///Check valve position
IF iq_stValve.i_xClsLS AND  iq_stValve.i_xOpnLS THEN
    iq_stValve.eState:=INVALID;
ELSIF NOT iq_stValve.i_xClsLS AND iq_stValve.i_xOpnLS AND iq_stValve.q_xOPN_DO THEN
    iq_stValve.eState:=OPEN;
ELSIF NOT iq_stValve.i_xClsLS AND iq_stValve.i_xOpnLS AND NOT iq_stValve.q_xOPN_DO THEN
    iq_stValve.eState:=OPEN_F;
ELSIF iq_stValve.i_xClsLS AND NOT iq_stValve.i_xOpnLS AND NOT iq_stValve.q_xOPN_DO THEN
    iq_stValve.eState:=CLOSED;
ELSIF NOT iq_stValve.i_xClsLS AND NOT iq_stValve.i_xOpnLS THEN
    iq_stValve.eState:=MOVING;
ELSE
    iq_stValve.eState:=INVALID;
END_IF

// Update hysteresis
///////////////////////////////////////////////////
IF iq_stValve.rAT_VAC_SP_LAST <> iq_stValve.rAT_VAC_SP OR xFirstPass THEN
    iq_stValve.rAT_VAC_SP_LAST := iq_stValve.rAT_VAC_SP;
    iq_stValve.rAT_VAC_HYS := iq_stValve.rHYST_PERC * iq_stValve.rAT_VAC_SP;
END_IF

iq_stValve.rAT_VAC_HYS := LIMIT(0, iq_stValve.rAT_VAC_HYS, iq_stValve.rAT_VAC_SP);
IF iq_stValve.rAT_VAC_SP <> 0 THEN
    IF iq_stValve.rHYST_PERC <> (iq_stValve.rAT_VAC_HYS / iq_stValve.rAT_VAC_SP) THEN
        iq_stValve.rHYST_PERC := LIMIT(0, (iq_stValve.rAT_VAC_HYS / iq_stValve.rAT_VAC_SP) ,1);
    END_IF

END_IF
// Valve at vacuum check
///////////////////////////////////////////////////
    set := i_stUSG.rPRESS < iq_stValve.rAT_VAC_HYS AND i_stDSG.rPRESS < iq_stValve.rAT_VAC_HYS AND i_stUSG.xPRESS_OK AND i_stDSG.xPRESS_OK;
     iq_stValve.xAT_VAC S= set;
    reset := i_stUSG.rPRESS > iq_stValve.rAT_VAC_SP OR i_stDSG.rPRESS > iq_stValve.rAT_VAC_SP OR NOT i_stUSG.xPRESS_OK OR NOT i_stDSG.xPRESS_OK;
    iq_stValve.xAT_VAC R= reset;

// Differential pressure check
///////////////////////////////////////////////////
    (* Calc the differential pressure across the valve *)
    rDiffPress := ABS(i_stUSG.rPRESS - i_stDSG.rPRESS);

    (* As long as the differential pressure is less than 30mbar, the valve is allowed to open *)
    IF rDiffPress <= rDiffPressAllowed AND i_stUSG.xPRESS_OK AND i_stDSG.xPRESS_OK THEN
        iq_stValve.xDP_OK := TRUE;
    ELSE
        iq_stValve.xDP_OK	:= FALSE;
        (* If the differential pressure is exceeded, even when the valve is open,
        the state is unexpected and triggers a fault, because it suggests that something
        is wrong with the valve, or gauges or mapping or there is a major leak on one side.*)
        iq_stValve.eVGC_State := ERR_DiffPress;
    END_IF

// Valve state
///////////////////////////////////////////////////
CASE iq_stValve.eVGC_State OF
    Vented: (* The Vented state is used during pump down *)
        //Log new state
        IF ePrevState <> iq_stValve.eVGC_State THEN
            fbLogger(sMsg:='Vented', eSevr:=TcEventSeverity.Info);
            ePrevState := iq_stValve.eVGC_State;
        END_IF

        (* Assuming the pump down went well, we are now at vacuum on both sides,
        so we move to the vacuum state, otherwise remain in the vented state *)
        IF iq_stValve.xAT_VAC AND (NOT (iq_stValve.xERR_DifPres)) AND  (NOT (iq_stValve.xERR_SP)) and  (NOT (iq_stValve.xERR_ExtFault))THEN
            iq_stValve.eVGC_State := AtVacuum;
        ELSE
            iq_stValve.eVGC_State := Vented;
        END_IF

    AtVacuum:
        //Log new state
        IF ePrevState <> iq_stValve.eVGC_State THEN
            fbLogger(sMsg:='Vacuum setpoint satisfied', eSevr:=TcEventSeverity.Info);
            ePrevState := iq_stValve.eVGC_State;
        END_IF

        IF iq_stValve.xAT_VAC THEN
        (* If both pressure setpoints are made,
        then enable the differential pressure interlock, regardless of the valve state
        assuming we're using some kind of ion gauge where a pressure setpoint cannot be higher than 1E-4 T *)
        iq_stValve.eVGC_State := AtVacuum;

        ELSE

            (* If the valve is open (or in an unknown state) and either gauge is not at it's vacuum setpoint,
            we have a loss of vacuum error *)
            IF (iq_stValve.i_xOpnLS OR (NOT iq_stValve.i_xOpnLS AND NOT iq_stValve.i_xClsLS)) THEN
                iq_stValve.eVGC_State := ERR_LostVac;
                iq_stValve.xERR_SP := TRUE; //TAW changed this to the ERR_SP bool because I think that's what it was intended to be?

            (* Alternatively, if the valve is already closed and we lose pressure on one side,
            it was probably intentional venting, so we calmly move back to venting mode, and
            disable the differential pressure interlock *) //??
            ELSIF iq_stValve.i_xClsLS THEN
                iq_stValve.eVGC_State := Vented;
            END_IF

        END_IF
    ERR_DiffPress:
        //Log new state
        IF ePrevState <> iq_stValve.eVGC_State THEN
            fbLogger(sMsg:='Potential accidental vent.', eSevr:=TcEventSeverity.Critical);
            ePrevState := iq_stValve.eVGC_State;
        END_IF

        IF NOT (iq_stValve.xERR_DifPres) THEN
            iq_stValve.eVGC_State := Vented;
        END_IF


    ERR_LostVac:
        //Log new state
        IF ePrevState <> iq_stValve.eVGC_State THEN
            fbLogger(sMsg:='Unexpected loss of vacuum while valve was open.', eSevr:=TcEventSeverity.Critical);
            ePrevState := iq_stValve.eVGC_State;
        END_IF
        IF NOT (iq_stValve.xERR_SP) THEN
            iq_stValve.eVGC_State := Vented;
        END_IF

    ERR_ExtFault:
        //Log new state
        IF ePrevState <> iq_stValve.eVGC_State THEN
            fbLogger(sMsg:='Lost external interlock while valve was open.', eSevr:=TcEventSeverity.Critical);
            ePrevState := iq_stValve.eVGC_State;
        END_IF
        IF NOT (iq_stValve.xERR_ExtFault) AND (NOT i_xExt_OK) THEN
            iq_stValve.eVGC_State := Vented;
        END_IF
    END_CASE



IF (NOT i_xExt_OK) THEN
    iq_stValve.eVGC_State := ERR_ExtFault;
    iq_stValve.xERR_ExtFault := TRUE;
END_IF

// Interlock evaluation - with bypass for DP ILK bypass
///////////////////////////////////////////////
IF i_xDis_DPIlk THEN
    iq_stValve.xOPN_OK := iq_stValve.xEXT_OK; // AND iq_stValve.xDP_OK ;
ELSE
    iq_stValve.xOPN_OK := iq_stValve.xEXT_OK AND iq_stValve.xAT_VAC;
END_IF


(* Valve operation *)

(* Override logic *)
(* Goal: give ability to override, but do so in a way that people won't forget it.
Solution: Override only after ten seconds of override, protect against blips,
when the valve permission goes true for more than ten seconds consistently, remove override
*)

tonDelOK(IN:=iq_stValve.xOPN_OK, PT:=tDelOK);
rtOK(CLK:=tonDelOK.Q);
IF rtOK.Q AND iq_stValve.pv_xOvrdOpn THEN
    iq_stValve.pv_xOvrdOpn :=FALSE;
    if (iq_stValve.eState = OPEN) AND (i_xOverrideMode) THEN iq_stValve.pv_xOPN_SW := TRUE; END_IF  //for seamless transition
    //Log
    fbLogger(sMsg:='Override expired', eSevr:=TcEventSeverity.Warning);

END_IF

//Override timer
tonOvrd(IN:=iq_stValve.pv_xOvrdOpn, PT:=tOvrd);

(* If Epics Command to close the Valve, check if PMPS and EPS are ok, otherwise Keep command set to open valve *)
IF NOT(iq_stValve.pv_xOPN_SW) AND ((NOT i_xPMPS_OK) OR (NOT i_xEPS_OK)) THEN
    //iq_stValve.pv_xOPN_SW := TRUE; // plc to only reset never to set this signal
END_IF
(* Reset the EPICS command to open the valve if the interlock is lost *)
(* based on EPS ok state, EPS overrides OPN_OK*)
IF NOT iq_stValve.xOPN_OK THEN
    IF i_xEPS_OK THEN iq_stValve.pv_xOPN_SW := FALSE; iq_stValve.sErrorMessage := 'ILK Active';
    ELSE //iq_stValve.pv_xOPN_SW := TRUE;		// plc to only reset never to set this signal
    END_IF
END_IF

(* Here's where the valve opens *)
iq_stValve.q_xOPN_DO := (iq_stValve.pv_xOPN_SW AND iq_stValve.xOPN_OK) OR (tonOvrd.Q AND i_xOverrideMode);

(* When the valve  is open MPS is OK*)
xMPS_OK := i_xOpnLS XOR i_xClsLS;

///Check valve moving postion timout
IF NOT iq_stValve.i_xClsLS AND tCLStimeout.Q THEN
    iq_stValve.bErrorPresent := TRUE;
    iq_stValve.sErrorMessage := 'Close Timeout';
ELSIF NOT iq_stValve.i_xOpnLS AND tOPNtimeout.Q THEN
    iq_stValve.bErrorPresent := TRUE;
    iq_stValve.sErrorMessage := 'Open Timeout';
END_IF
IF (iq_stValve.eState=INVALID) THEN
    iq_stValve.bErrorPresent := TRUE;
    iq_stValve.sErrorMessage := CONCAT(sPath,'Invalid Valve Position');
END_IF
(*Timers*)
tOPNtimeout(IN:= iq_stValve.q_xOPN_DO, PT := tTimeOutDuration );
tCLStimeout(IN:= NOT iq_stValve.q_xOPN_DO, PT := tTimeOutDuration);


// Log valve timeouts
tErrorPresent(CLK:=iq_stValve.bErrorPresent);
IF tErrorPresent.Q THEN fbLogger(sMsg:=iq_stValve.sErrorMessage, eSevr:=TcEventSeverity.Warning); END_IF

// Log valve open
tAction(CLK:= iq_stValve.q_xOPN_DO);
IF tAction.Q THEN fbLogger(sMsg:='Valve commanded open', eSevr:=TcEventSeverity.Info); END_IF

// Log override mode enabled
tOverrideActivated(CLK:= (tonOvrd.Q AND i_xOverrideMode));
IF tOverrideActivated.Q THEN fbLogger(sMsg:='Valve override mode activated', eSevr:=TcEventSeverity.Warning); END_IF


// Alarm reset
//////////////////////////////////////
ACT_ResetAlarms();

(*IO Mapping*)
ACT_IO();

(*FAST FAULT*)
fbFF(i_xOK := xMPS_OK,
    i_xReset := i_xReset,
    i_xAutoReset :=TRUE,
    io_fbFFHWO := io_fbFFHWO);

ACTION ACT_IO:
(*inputs*)
iq_stValve.i_xOpnLS := 	i_xOpnLS;
iq_stValve.i_xClsLS:=	i_xClsLS;
iq_stValve.xEXT_OK := i_xEXT_OK;
iq_stValve.xOverrideMode := i_xOverrideMode;
(*outputs*)
q_xOPN_DO:= iq_stValve.q_xOPN_DO;
END_ACTION

ACTION ACT_ResetAlarms:
iq_stValve.xERR_DifPres R= iq_stValve.pv_xAlmRst;
iq_stValve.xERR_SP R= iq_stValve.pv_xAlmRst;
iq_stValve.bErrorPresent R= iq_stValve.pv_xAlmRst;

IF ( iq_stValve.pv_xAlmRst) THEN
    iq_stValve.sErrorMessage :='';
END_IF
END_ACTION

METHOD PUBLIC M_IsClosed : BOOL
VAR_INPUT
END_VAR
M_IsClosed := (This^.iq_stValve.eState = E_ValvePositionState.CLOSED);
END_METHOD

METHOD PUBLIC M_IsOpen : BOOL
VAR_INPUT
END_VAR
M_IsOpen := (This^.iq_stValve.eState = E_ValvePositionState.OPEN);
END_METHOD

// Use this Methode to Open or close the valve by setting the OPN_SW to the input value.
METHOD PUBLIC M_Set_OPN_SW : BOOL
VAR_INPUT
        value:BOOL;
END_VAR
This^.iq_stValve.pv_xOPN_SW := value;
END_METHOD

END_FUNCTION_BLOCK

// ---- POUs/Functions/Deprecated/Valves/FB_VGC_EBD.TcPOU
(*Deprecated*)
(* This function block is similar to the FB_VGC, except it has 2 outputs to actuate the Valve*)
(* This function block implements basic functionality for Isolation Gate Valves*)
(* This function block interlock is as follows:
1. The valve can be opened when the difference between the pressures on both sides is
less than the maximum differential pressure.
2. This rule persists until the pressures on both sides are lower than the vacuum-setpoint.
3. Once at-vac, the valve will close if the pressure on either side rises above the setpoint.*)
(*This function block also implements PMPS and EPS interlocks, as well as Fast MPS trigger*)
{attribute 'no_check'}
{attribute 'obsolete' := 'FB_VGC_EBD has been deprecated and is not valid!'}
FUNCTION_BLOCK FB_VGC_EBD
VAR_IN_OUT

END_VAR
VAR_INPUT
    (*Upstream Gauge, usually ion gauge*)
    i_stUSG	:	ST_VG;
    (*Downstream Gauge, usually ion gauge*)
    i_stDSG	:	ST_VG;
    {attribute 'pytmc' := '
    pv: Dis_DPIlk
    '}
    i_xDis_DPIlk : BOOL := FALSE;  (* Set to true when calling the function to disable the differential pressure interlock *)
    {attribute 'pytmc' := '
    pv: EPS_OK
    '}
    i_xEPS_OK:	BOOL	:= TRUE; (*External EPS interlock, Set to TRUE when no EPS interlock is required, otherwise set to correct interlock signal*)
    {attribute 'pytmc' := '
    pv: MPS_OK
    '}
    i_xPMPS_OK:	BOOL	; (*External MPS interlock, Set to TRUE when no PMPS interlock is required*)
    i_xExt_OK: BOOL; (*Other External Interlock, Set to True when no external interlock is required*)
    i_xOverrideMode : BOOL; (*To be linked to global override bit. This Overrides Vacuum logic only, EPS, MPS and PMPS are still enforces*)
    // Reset fault
    {attribute 'pytmc' := '
    pv: FF_Reset
    '}
    i_xReset: BOOL;
    i_sDevName : T_MaxString :=  'VGC'; // Device name for diagnostic
END_VAR
VAR_OUTPUT
    {attribute 'pytmc' := '
    pv:
    '}
    iq_stValve : ST_VGC; (* All valve data and states will be in this struct*)

    {attribute 'pytmc' := '
    pv: MPS_FAULT_OK
    field: ZNAM MPS FAULT ;
    field: ONAM MPS OK ;
    '}
    xMPS_OK:	BOOL; (*MPS Fast OK, is set when the Valve is Open*)
END_VAR
VAR_IN_OUT
    io_fbFFHWO    :    FB_HardwareFFOutput;
END_VAR
VAR
    // PMPS
    fbFF    :    FB_FastFault :=(
        i_DevName := 'VGC',
        i_Desc := 'Fault occurs when the valve is not in open state',
        i_TypeCode := 16#1010);
    {attribute 'instance-path'}
    {attribute 'noinit'}
    sPath: STRING;

    rDiffPressAllowed	:	REAL := 22.5; // Torr, Default value comes from Vat Valve Manual
    rDiffPress : REAL;
    set : BOOL;
    reset: BOOL;

    xFirstPass	:	BOOL;
    fbFSInit		:	R_TRIG;

    tonDelOK : TON;
    rtOK	:	R_TRIG;
    tonOvrd	:	TON;

    tDelOK	:	TIME := T#60S;
    tOvrd	:	TIME := T#10s;


    (* Timeouts*)
    tTimeOutDuration: TIME:= T#30S;
    tOPNtimeout: TON;
    tCLStimeout:TON;


     // For logging
    fbLogger : FB_LogMessage := (eSubsystem:=E_SubSystem.VACUUM);
    ePrevState : E_VGC;
    tErrorPresent : R_TRIG;
    tAction : R_TRIG; // Primary action of this device (OPN_DO, PUMP_RUN, etc.)
    tOverrideActivated : R_TRIG;

    (*IO*)
    i_xOpnLS	AT%I*: BOOL;
    i_xClsLS	AT%I*: BOOL;
    q_xOPN_DO	AT%Q*: BOOL;
    q_xOPN_DO_2	AT%Q*: BOOL;

END_VAR

(* Vacuum gate valve
A. Wallace
16-10-29

A gate valve isolates vacuum volumes. Ideally it can be opened when a system is vented
to allow for faster pumping, and will close when high vacuum is lost.

The following behavior is good for valves in something like a gas attenuator.
This function block does the following:
1. The valve can be opened when the difference between the pressures on both sides is
less than the maximum differential pressure.
2. This rule persists until the pressures on both sides are lower than the vacuum-setpoint.
3. Once at-vac, the valve will close if the pressure on either side rises above the setpoint.

Alternatively, the differential pressure interlock can be disabled so the valve may only be opened
if the pressure on both sides is lower than the at-vacuum-setpoint. You want this behavior if
the valve is to be used in a UHV section.

Hysteresis is employed to ensure a smooth transition from vented/pumping down, to at-vac.

Finally, an override system is built in so you can bypass all the interlocking logic and
get back online.
*)
(* 10/1/2018 Margaret Ghaly included EPS, PMPS Checkes and MPS trigger signals*)


fbFSInit( CLK := TRUE, Q => xFirstPass);
(*IO Mapping*)
ACT_IO();

(* On first PLC pass, put valve into vented state, which implies a closed valve *)
IF xFirstPass THEN
    iq_stValve.eVGC_State := Vented;
    iq_stValve.pv_xOPN_SW := FALSE;
    fbFF.i_DevName := i_sDevName;
END_IF


///Check valve postion
IF iq_stValve.i_xClsLS AND  iq_stValve.i_xOpnLS THEN
    iq_stValve.eState:=INVALID;
ELSIF NOT iq_stValve.i_xClsLS AND iq_stValve.i_xOpnLS AND iq_stValve.q_xOPN_DO THEN
    iq_stValve.eState:=OPEN;
ELSIF iq_stValve.i_xClsLS AND NOT iq_stValve.i_xOpnLS AND NOT iq_stValve.q_xOPN_DO THEN
    iq_stValve.eState:=CLOSED;
ELSIF NOT iq_stValve.i_xClsLS AND NOT iq_stValve.i_xOpnLS THEN
    iq_stValve.eState:=MOVING;
ELSE
    iq_stValve.eState:=INVALID;
END_IF

// Update hysteresis
///////////////////////////////////////////////////
IF iq_stValve.rAT_VAC_SP_LAST <> iq_stValve.rAT_VAC_SP OR xFirstPass THEN
    iq_stValve.rAT_VAC_SP_LAST := iq_stValve.rAT_VAC_SP;
    iq_stValve.rAT_VAC_HYS := iq_stValve.rHYST_PERC * iq_stValve.rAT_VAC_SP;
END_IF

iq_stValve.rAT_VAC_HYS := LIMIT(0, iq_stValve.rAT_VAC_HYS, iq_stValve.rAT_VAC_SP);
IF iq_stValve.rAT_VAC_SP <> 0 THEN
    IF iq_stValve.rHYST_PERC <> (iq_stValve.rAT_VAC_HYS / iq_stValve.rAT_VAC_SP) THEN
        iq_stValve.rHYST_PERC := LIMIT(0, (iq_stValve.rAT_VAC_HYS / iq_stValve.rAT_VAC_SP) ,1);
    END_IF

END_IF
// Valve at vacuum check
///////////////////////////////////////////////////
    set := i_stUSG.rPRESS < iq_stValve.rAT_VAC_HYS AND i_stDSG.rPRESS < iq_stValve.rAT_VAC_HYS AND i_stUSG.xPRESS_OK AND i_stDSG.xPRESS_OK;
     iq_stValve.xAT_VAC S= set;
    reset := i_stUSG.rPRESS > iq_stValve.rAT_VAC_SP OR i_stDSG.rPRESS > iq_stValve.rAT_VAC_SP OR NOT i_stUSG.xPRESS_OK OR NOT i_stDSG.xPRESS_OK;
    iq_stValve.xAT_VAC R= reset;

// Differential pressure check
///////////////////////////////////////////////////
    (* Calc the differential pressure across the valve *)
    rDiffPress := ABS(i_stUSG.rPRESS - i_stDSG.rPRESS);

    (* As long as the differential pressure is less than 30mbar, the valve is allowed to open *)
    IF rDiffPress <= rDiffPressAllowed AND i_stUSG.xPRESS_OK AND i_stDSG.xPRESS_OK THEN
        iq_stValve.xDP_OK := TRUE;
    ELSE
        iq_stValve.xDP_OK	:= FALSE;
        (* If the differential pressure is exceeded, even when the valve is open,
        the state is unexpected and triggers a fault, because it suggests that something
        is wrong with the valve, or gauges or mapping or there is a major leak on one side.*)
        iq_stValve.eVGC_State := ERR_DiffPress;
        iq_stValve.xERR_DifPres := TRUE;
    END_IF

// Valve state
///////////////////////////////////////////////////
CASE iq_stValve.eVGC_State OF
    Vented: (* The Vented state is used during pump down *)
        //Log new state
        IF ePrevState <> iq_stValve.eVGC_State THEN
            fbLogger(sMsg:='Vented', eSevr:=TcEventSeverity.Info);
            ePrevState := iq_stValve.eVGC_State;
        END_IF

        (* Assuming the pump down went well, we are now at vacuum on both sides,
        so we move to the vacuum state, otherwise remain in the vented state *)
        IF iq_stValve.xAT_VAC AND (NOT (iq_stValve.xERR_DifPres)) AND  (NOT (iq_stValve.xERR_SP)) and  (NOT (iq_stValve.xERR_ExtFault))THEN
            iq_stValve.eVGC_State := AtVacuum;
        ELSE
            iq_stValve.eVGC_State := Vented;
        END_IF

    AtVacuum:
        //Log new state
        IF ePrevState <> iq_stValve.eVGC_State THEN
            fbLogger(sMsg:='Vacuum setpoint satisfied', eSevr:=TcEventSeverity.Info);
            ePrevState := iq_stValve.eVGC_State;
        END_IF

        IF iq_stValve.xAT_VAC THEN
        (* If both pressure setpoints are made,
        then enable the differential pressure interlock, regardless of the valve state
        assuming we're using some kind of ion gauge where a pressure setpoint cannot be higher than 1E-4 T *)
        iq_stValve.eVGC_State := AtVacuum;

        ELSE

            (* If the valve is open (or in an unknown state) and either gauge is not at it's vacuum setpoint,
            we have a loss of vacuum error *)
            IF (iq_stValve.i_xOpnLS OR (NOT iq_stValve.i_xOpnLS AND NOT iq_stValve.i_xClsLS)) THEN
                iq_stValve.eVGC_State := ERR_LostVac;
                iq_stValve.xERR_SP := TRUE; //TAW changed this to the ERR_SP bool because I think that's what it was intended to be?

            (* Alternatively, if the valve is already closed and we lose pressure on one side,
            it was probably intentional venting, so we calmly move back to venting mode, and
            disable the differential pressure interlock *) //??
            ELSIF iq_stValve.i_xClsLS THEN
                iq_stValve.eVGC_State := Vented;
            END_IF

        END_IF

    ERR_DiffPress:
        //Log new state
        IF ePrevState <> iq_stValve.eVGC_State THEN
            fbLogger(sMsg:='Potential accidental vent.', eSevr:=TcEventSeverity.Critical);
            ePrevState := iq_stValve.eVGC_State;
        END_IF

        IF NOT (iq_stValve.xERR_DifPres) THEN
            iq_stValve.eVGC_State := Vented;
        END_IF


    ERR_LostVac:
        //Log new state
        IF ePrevState <> iq_stValve.eVGC_State THEN
            fbLogger(sMsg:='Unexpected loss of vacuum while valve was open.', eSevr:=TcEventSeverity.Critical);
            ePrevState := iq_stValve.eVGC_State;
        END_IF
        IF NOT (iq_stValve.xERR_SP) THEN
            iq_stValve.eVGC_State := Vented;
        END_IF

    ERR_ExtFault:
        //Log new state
        IF ePrevState <> iq_stValve.eVGC_State THEN
            fbLogger(sMsg:='Lost external interlock while valve was open.', eSevr:=TcEventSeverity.Critical);
            ePrevState := iq_stValve.eVGC_State;
        END_IF
        IF NOT (iq_stValve.xERR_ExtFault) AND (NOT i_xExt_OK) THEN
            iq_stValve.eVGC_State := Vented;
        END_IF
END_CASE

IF (NOT i_xExt_OK) THEN
    iq_stValve.eVGC_State := ERR_ExtFault;
    iq_stValve.xERR_ExtFault := TRUE;
END_IF

// Interlock evaluation - with bypass for DP ILK bypass
///////////////////////////////////////////////
IF i_xDis_DPIlk THEN
    iq_stValve.xOPN_OK := iq_stValve.xEXT_OK; // AND iq_stValve.xDP_OK ;
ELSE
    iq_stValve.xOPN_OK := iq_stValve.xEXT_OK AND iq_stValve.xAT_VAC;
END_IF


(* Valve operation *)

(* Override logic *)
(* Goal: give ability to override, but do so in a way that people won't forget it.
Solution: Override only after ten seconds of override, protect against blips,
when the valve permission goes true for more than ten seconds consistently, remove override
*)

tonDelOK(IN:=iq_stValve.xOPN_OK, PT:=tDelOK);
rtOK(CLK:=tonDelOK.Q);
IF rtOK.Q AND iq_stValve.pv_xOvrdOpn THEN
    iq_stValve.pv_xOvrdOpn :=FALSE;
    if (iq_stValve.eState = OPEN) AND (i_xOverrideMode) THEN iq_stValve.pv_xOPN_SW := TRUE; END_IF //for seamless transition
    //Log
    fbLogger(sMsg:='Override expired', eSevr:=TcEventSeverity.Warning);

END_IF

//Override timer
tonOvrd(IN:=iq_stValve.pv_xOvrdOpn, PT:=tOvrd);

(* If Epics Command to close the Valve, check if PMPS and EPS are ok, otherwise Keep command set to open valve *)
IF NOT(iq_stValve.pv_xOPN_SW) AND ((NOT i_xPMPS_OK) OR (NOT i_xEPS_OK)) THEN
    //iq_stValve.pv_xOPN_SW := TRUE; // plc to only reset never to set this signal
END_IF
(* Reset the EPICS command to open the valve if the interlock is lost *)
(* based on EPS ok state, EPS overrides OPN_OK*)
IF NOT iq_stValve.xOPN_OK THEN
    IF i_xEPS_OK THEN iq_stValve.pv_xOPN_SW := FALSE; iq_stValve.sErrorMessage := 'ILK Active';
    ELSE //iq_stValve.pv_xOPN_SW := TRUE;		// plc to only reset never to set this signal
    END_IF
END_IF

(* Here's where the valve opens *)
iq_stValve.q_xOPN_DO := (iq_stValve.pv_xOPN_SW AND iq_stValve.xOPN_OK) OR (tonOvrd.Q AND i_xOverrideMode);

(* When the valve  is open MPS is OK*)
xMPS_OK := (iq_stValve.eState=OPEN) OR (iq_stValve.eState=OPEN_F);//iq_stValve.i_xOpnLS;

///Check valve moving postion timout
IF NOT iq_stValve.i_xClsLS AND tCLStimeout.Q THEN
    iq_stValve.bErrorPresent := TRUE;
    iq_stValve.sErrorMessage := ' Close Timeout';
ELSIF NOT iq_stValve.i_xOpnLS AND tOPNtimeout.Q THEN
    iq_stValve.bErrorPresent := TRUE;
    iq_stValve.sErrorMessage := ' Open Timeout';
END_IF
IF (iq_stValve.eState=INVALID) THEN
    iq_stValve.bErrorPresent := TRUE;
    iq_stValve.sErrorMessage := CONCAT(sPath,' Invalid Valve Position');
END_IF


(*Timers*)
tOPNtimeout(IN:= iq_stValve.q_xOPN_DO, PT := tTimeOutDuration );
tCLStimeout(IN:= NOT iq_stValve.q_xOPN_DO, PT := tTimeOutDuration);

// Log valve timeouts
tErrorPresent(CLK:=iq_stValve.bErrorPresent);
IF tErrorPresent.Q THEN fbLogger(sMsg:=iq_stValve.sErrorMessage, eSevr:=TcEventSeverity.Warning); END_IF

// Log valve open
tAction(CLK:= iq_stValve.q_xOPN_DO);
IF tAction.Q THEN fbLogger(sMsg:='Valve commanded open', eSevr:=TcEventSeverity.Info); END_IF

// Log override mode enabled
tOverrideActivated(CLK:= (tonOvrd.Q AND i_xOverrideMode));
IF tOverrideActivated.Q THEN fbLogger(sMsg:='Valve override mode activated', eSevr:=TcEventSeverity.Warning); END_IF

// Alarm reset
//////////////////////////////////////
ACT_ResetAlarms();

(*IO Mapping*)
ACT_IO();

(*FAST FAULT*)
fbFF(i_xOK := xMPS_OK,
    i_xReset := i_xReset,
    i_xAutoReset :=TRUE,
    io_fbFFHWO := io_fbFFHWO);

ACTION ACT_IO:
(*inputs*)
iq_stValve.i_xOpnLS := 	i_xOpnLS;
iq_stValve.i_xClsLS:=	i_xClsLS;
iq_stValve.xEXT_OK := i_xEXT_OK;
iq_stValve.xOverrideMode := i_xOverrideMode;
(*outputs*)
q_xOPN_DO:= iq_stValve.q_xOPN_DO;
q_xOPN_DO_2:= iq_stValve.q_xOPN_DO;


(*ILK Devices*)
iq_stValve.sIlkUSDeviceName := This^.i_stUSG.sPath;
iq_stValve.sIlkDSDeviceName := This^.i_stDSG.sPath;
END_ACTION

ACTION ACT_ResetAlarms:
iq_stValve.xERR_DifPres R= iq_stValve.pv_xAlmRst;
iq_stValve.xERR_SP R= iq_stValve.pv_xAlmRst;
iq_stValve.bErrorPresent R= iq_stValve.pv_xAlmRst;

IF ( iq_stValve.pv_xAlmRst) THEN
    iq_stValve.sErrorMessage :='';
END_IF
END_ACTION

METHOD PUBLIC M_IsClosed : BOOL
VAR_INPUT
END_VAR
M_IsClosed := (This^.iq_stValve.eState = E_ValvePositionState.CLOSED);
END_METHOD

METHOD PUBLIC M_IsOpen : BOOL
VAR_INPUT
END_VAR
M_IsOpen := (This^.iq_stValve.eState = E_ValvePositionState.OPEN);
END_METHOD

// Use this Methode to Open or close the valve by setting the OPN_SW to the input value.
METHOD PUBLIC M_Set_OPN_SW : BOOL
VAR_INPUT
        value:BOOL;
END_VAR
This^.iq_stValve.pv_xOPN_SW := value;
END_METHOD

END_FUNCTION_BLOCK

// ---- POUs/Functions/Gauges/FB_901_ECAT.TcPOU
(* works for 901 with Ethercat interface*)
{attribute 'no_check'}
FUNCTION_BLOCK FB_901_ECAT  EXTENDS FB_GaugeBase
VAR_INPUT
END_VAR
VAR_OUTPUT
    {attribute 'pytmc' := '
    pv:
    '}
    PG	: ST_VG;
END_VAR
VAR_IN_OUT

END_VAR
VAR
    bInit: BOOL:= TRUE;(*IO*)
    xPress_OK AT%I* : BOOL;
    xOverrange AT%I* : BOOL;
    xUnderrange AT%I* : BOOL;
    i_iPRESS_R AT%I* : REAL; // input Pressure // Link to analog Input
    bWcstate AT%I* : BOOL; // 0: date valid, 1: date invalid

END_VAR

(* Standard MKS 9XX series conversion *)
(* works for 901 with Ethercat interface*)
// no div by zero
PG.rPRESS :=i_iPRESS_R;
PG.xPRESS_OK := xPress_OK and NOT bWcstate ;
IF xPress_OK and NOT bWcstate THEN
    PG.xPRESS_OK := TRUE;
    PG.eState := Valid; //Press OK
ELSIF xOverrange and NOT bWcstate THEN
    PG.xPRESS_OK := FALSE;
    PG.eState := OoR;
ELSIF xUnderrange and NOT bWcstate THEN
    PG.xPRESS_OK := FALSE;
    PG.eState := PressInvalid;

END_IF



(*Logger*)
ACT_Logger();
(* Soft IO Mapping*)
ACT_IO();

ACTION ACT_Init:
IF (bInit) THEN
    bInit := False;

    //set pressure units to Torr
    // value 0x00A10000 SDO index 0xf840, si 0x01 UDINT
END_IF
END_ACTION

ACTION ACT_IO:

IF PG.xPRESS_OK THEN
      PG.i_iPRESS_R := REAL_TO_INT(i_iPRESS_R);
ELSE
    PG.rPRESS := 0.0;
END_IF
PG.sPath := sPath;
END_ACTION

ACTION ACT_Logger:

//STATE Logger
IF ePrevState <> PG.eState THEN
      CASE PG.eState OF
        ValidHi:
            fbLogger(sMsg:='Gauge pressure valid high.', eSevr:=TcEventSeverity.Info);
        ValidLo:
            fbLogger(sMsg:='Gauge pressure valid low.', eSevr:=TcEventSeverity.Info);
        Valid:
            fbLogger(sMsg:='Gauge pressure valid.', eSevr:=TcEventSeverity.Info);
          GaugeDisconnected:
            fbLogger(sMsg:='Gauge Disconnected.', eSevr:=TcEventSeverity.Critical);
        PressInvalid:
            fbLogger(sMsg:='Gauge pressure invalid.', eSevr:=TcEventSeverity.Warning);
        OoR:
            fbLogger(sMsg:='Gauge pressure out of range.', eSevr:=TcEventSeverity.Warning);
        Starting:
            fbLogger(sMsg:='Gauge starting.', eSevr:=TcEventSeverity.Info);
      END_CASE
      ePrevState := PG.eState;
  END_IF
END_ACTION

END_FUNCTION_BLOCK

// ---- POUs/Functions/Gauges/FB_9XX.TcPOU
(* Standard MKS 9XX series conversion *)
(* works for 925 *)
FUNCTION_BLOCK FB_9XX EXTENDS FB_GaugeBase
VAR_INPUT
END_VAR
VAR_OUTPUT
    {attribute 'pytmc' := '
    pv:
    '}
    PG	: ST_VG;
END_VAR
VAR_IN_OUT
END_VAR
VAR
    rV : REAL;
    fbGaugeState : FB_PressureState;
    rMaxPressure	:	REAL := 760; //Torr
    rMinPressure	:	REAL := 1E-5; //Torr
    rVMin : REAL:= 0.9;

    iTermBits: UINT := 30518 ; // The terminal's maximum value in bits default el3174 as per vacuum architecture
    (*IO*)
    i_iPRESS_R AT%I* :INT; // input Pressure // Link to analog Input
END_VAR

VAR CONSTANT
    (*Default set point 50 mT*)
    rDefaultVAC_SP: REAL := 5E-2;
END_VAR

(* Standard MKS 9XX series conversion *)
(* works for 972 and 925 *)


//Default setpoint
IF PG.rVAC_SP = 0 THEN
    PG.rVAC_SP := rDefaultVAC_SP;
END_IF
// check no div by zero
If (iTermBits=0) THEN iTermBits := 30518;END_IF
rV := 10*INT_TO_REAL(PG.i_iPRESS_R)/iTermBits;

IF rV >=rVMin THEN
    IF rV >= rVMin AND rV <= 1 THEN
        PG.rPRESS := 1E-5;
    ELSE
        PG.rPRESS := LREAL_TO_REAL(EXPT(10, rV-6));
    END_IF
    PG.xPRESS_OK := TRUE;
    PG.eState := Valid;
ELSE
    PG.xPRESS_OK := FALSE;
    IF (rV = 0) THEN PG.eState := GaugeDisconnected;
        ELSE  PG.eState := PressInvalid;
    END_IF
END_IF

(* Setpoint evaluation *)
PG.xAT_VAC := PG.xPRESS_OK AND (PG.rPRESS < PG.rVAC_SP);


(*Logger*)
ACT_Logger();
(*Soft IO Mapping*)
ACT_IO();

ACTION ACT_IO:
PG.i_iPRESS_R :=i_iPRESS_R;
PG.sPath := sPath;
END_ACTION

ACTION ACT_Logger:

//STATE Logger
IF ePrevState <> PG.eState THEN
      CASE PG.eState OF
        ValidHi:
            fbLogger(sMsg:='Gauge pressure valid high.', eSevr:=TcEventSeverity.Info);
        ValidLo:
            fbLogger(sMsg:='Gauge pressure valid low.', eSevr:=TcEventSeverity.Info);
        Valid:
            fbLogger(sMsg:='Gauge pressure valid.', eSevr:=TcEventSeverity.Info);
          GaugeDisconnected:
            fbLogger(sMsg:='Gauge Disconnected.', eSevr:=TcEventSeverity.Critical);
        PressInvalid:
            fbLogger(sMsg:='Gauge pressure invalid.', eSevr:=TcEventSeverity.Warning);
        OoR:
            fbLogger(sMsg:='Gauge pressure out of range.', eSevr:=TcEventSeverity.Warning);
        Starting:
            fbLogger(sMsg:='Gauge starting.', eSevr:=TcEventSeverity.Info);
      END_CASE
      ePrevState := PG.eState;
  END_IF
END_ACTION

METHOD M_SetBits : BOOL
VAR_INPUT
    TermBits : UINT; // The terminal's maximum value in bits
END_VAR
This^.iTermBits := TermBits;
END_METHOD

END_FUNCTION_BLOCK

// ---- POUs/Functions/Gauges/FB_972.TcPOU
{attribute 'no_check'}
FUNCTION_BLOCK FB_972  EXTENDS FB_GaugeBase
VAR_INPUT
END_VAR
VAR_OUTPUT
    {attribute 'pytmc' := '
    pv:
    '}
    PG	: ST_VG;
END_VAR
VAR_IN_OUT

END_VAR
VAR
    rV : REAL;
    iTermBits: UINT := 32767 ; // The terminal's maximum value in bits
    (*IO*)
    i_iPRESS_R AT%I* :INT; // input Pressure // Link to analog Input
END_VAR

(* Standard MKS 9XX series conversion *)
(* works for 972 and 925 *)
// no div by zero
If (iTermBits=0) THEN iTermBits := 32767;END_IF
rV := 10*INT_TO_REAL(PG.i_iPRESS_R)/iTermBits;

IF (rV > 1) AND (rV <= 7) THEN
    PG.rPRESS := LREAL_TO_REAL(EXPT(10, 2*rV-11));
    PG.xPRESS_OK := TRUE;
    PG.eState := Valid; //Press OK
ELSE
    PG.xPRESS_OK := FALSE;
    IF (rV <= 1) THEN PG.eState := GaugeDisconnected;
        ELSE PG.eState := OoR;
    END_IF
END_IF

(* Setpoint evaluation *)
PG.xAT_VAC := PG.xPRESS_OK AND (PG.rPRESS < PG.rVAC_SP);

(*Logger*)
ACT_Logger();
(* Soft IO Mapping*)
ACT_IO();

ACTION ACT_IO:
PG.i_iPRESS_R :=i_iPRESS_R;
PG.sPath := sPath;
END_ACTION

ACTION ACT_Logger:

//STATE Logger
IF ePrevState <> PG.eState THEN
      CASE PG.eState OF
        ValidHi:
            fbLogger(sMsg:='Gauge pressure valid high.', eSevr:=TcEventSeverity.Info);
        ValidLo:
            fbLogger(sMsg:='Gauge pressure valid low.', eSevr:=TcEventSeverity.Info);
        Valid:
            fbLogger(sMsg:='Gauge pressure valid.', eSevr:=TcEventSeverity.Info);
          GaugeDisconnected:
            fbLogger(sMsg:='Gauge Disconnected.', eSevr:=TcEventSeverity.Critical);
        PressInvalid:
            fbLogger(sMsg:='Gauge pressure invalid.', eSevr:=TcEventSeverity.Warning);
        OoR:
            fbLogger(sMsg:='Gauge pressure out of range.', eSevr:=TcEventSeverity.Warning);
        Starting:
            fbLogger(sMsg:='Gauge starting.', eSevr:=TcEventSeverity.Info);
      END_CASE
      ePrevState := PG.eState;
  END_IF
END_ACTION

METHOD M_SetBits : BOOL
VAR_INPUT
    TermBits : UINT; // The terminal's maximum value in bits
END_VAR
This^.iTermBits := TermBits;
END_METHOD

END_FUNCTION_BLOCK

// ---- POUs/Functions/Gauges/FB_IE514.TcPOU
(*This function is for the IE514 connected to controller IM540*)
(*This function provides ILK and Set Point Protection for the IE514*)
FUNCTION_BLOCK FB_IE514 EXTENDS FB_GaugeBase
VAR_IN_OUT
END_VAR
VAR_INPUT
    PG : ST_VG;
END_VAR
VAR_OUTPUT
    {attribute 'pytmc' := '
        pv:01
    '}
    IG_CH1 : ST_VG;
    {attribute 'pytmc' := '
        pv:02
    '}
    IG_CH2 : ST_VG;
END_VAR
VAR
    rV_CH1 : REAL; //Raw value in volts for CH1 calculated from iTermBits
    rV_CH2 : REAL; //Raw value in volts for CH2 calculated from iTermBits

    tHvDis_CH1 : TON := (PT := T#20S); //HV turn on timer
    tHvDis_CH2 : TON := (PT := T#20S); //HV turn on timer

    rtHvSw_CH1 : R_TRIG;
    rtHvSw_CH2 : R_TRIG;

    tAction_CH1 : R_TRIG;
    tAction_CH2 : R_TRIG;

    ePrevStateIG_CH1 : E_PressureState;
    ePrevStateIG_CH2 : E_PressureState;

    //rDefaultVAC_SP: REAL := 9E-3; // as per manual

    iTermBits : UINT := 30518; // The terminal's maximum value in bits default el3174 as per vacuum architecture
    binit : BOOL := TRUE;  // Do something at startup

    (*IOs to be linked*)
    /// Controls and I/Os
    i_iPRESS_R_CH1 AT %I* : INT; // input raw pressure in bits CH1 (ADC) // 'TcLinkTo' (EL3174) ^Input
    i_iPRESS_R_CH2 AT %I* : INT; // input raw pressure in bits CH2 (ADC) // 'TcLinkTo' (EL3174) ^Input
    q_xHV_DIS_CH1 AT %Q* : BOOL; // Enable Gauge High Voltage on CH1 when True // 'TcLinkTo' (EL2124) ^Output
    q_xHV_DIS_CH2 AT %Q* : BOOL; // Enable Gauge High Voltage on CH2 when True // 'TcLinkTo' (EL2124) ^Output
    i_xHV_ON AT %I*	: BOOL; // True when EMI is on  // 'TcLinkTo' (EL1004 or EL1008) ^Input
    i_xERR_CH1 AT %I* : BOOL; // TRUE when NO error is present on assigned channel
    i_xERR_CH2 AT %I* : BOOL; // TRUE when NO error is present on assigned channel
    i_xCH2_SEL AT %I* : BOOL; // TRUE when CH2 selected, FALSE when CH1 selected
END_VAR
VAR CONSTANT
    cMaxPressure : REAL := 7.5E-5; //Torr
    cMinPressure : REAL := 7.5E-14; //Torr
    cGaugeMinVoltage : REAL := 1.111; //minimum voltage corresponds to 7.5E-13 (7.498E-13)Torr which should be the minimum pressure IE514 can read.
    cGaugeMaxVoltage : REAL := 10.0; //maximum voltage corresponds 7.5E-5 Torr which should be the maximum pressure IE514 can read.
    cGaugeDisconnected : REAL := 10.2; //voltage when gauge is disconnected.
    cGaugeOff : REAL := 10.2; //voltage when gauge is turned off
    cDeadband : REAL := 0.05; //deadband in voltage
END_VAR
VAR PERSISTENT
    //Persistent variables for CH1
    rVAC_SP_CH1 : REAL;
    rPRO_SP_CH1 : REAL;
    rHYS_PR_CH1 : REAL;
    //Persistent variables for CH2
    rVAC_SP_CH2 : REAL;
    rPRO_SP_CH2 : REAL;
    rHYS_PR_CH2 : REAL;
END_VAR

(* 2-6-2023, Janez Govednik *)
(* This function will read the pressure from an IE514 gauge on an IM540. *)

(*Only ONE channel can be turned ON at the same time*)
rtHvSw_CH1(CLK := IG_CH1.xHV_SW);
rtHvSw_CH2(CLK := IG_CH2.xHV_SW);
IF rtHvSw_CH1.Q THEN
    IG_CH2.xHV_SW := FALSE;
    IG_CH2.q_xHV_DIS := FALSE;
END_IF

IF rtHvSw_CH2.Q THEN
    IG_CH1.xHV_SW := FALSE;
    IG_CH1.q_xHV_DIS := FALSE;
END_IF

//Start timers when HV ON signal triggered
tHvDis_CH1(IN := IG_CH1.q_xHV_DIS, Q => IG_CH1.xTurnOnTime);
tHvDis_CH2(IN := IG_CH2.q_xHV_DIS, Q => IG_CH2.xTurnOnTime);

(*Raw voltage conversion*)
//check no div by zero
IF (iTermBits = 0) THEN iTermBits := 30518; END_IF
rV_CH1 := 10*INT_TO_REAL(i_iPRESS_R_CH1)/iTermBits;
rV_CH2 := 10*INT_TO_REAL(i_iPRESS_R_CH2)/iTermBits;

(*RAW voltage to Pressure conversion*)
IG_CH1.rPRESS := LREAL_TO_REAL(EXPT(10, rV_CH1/10*LOG(cMaxPressure/cMinPressure) + LOG(cMinPressure))); //manual page 70 IM540 (Mode Full), (Scale) = Log
IG_CH2.rPRESS := LREAL_TO_REAL(EXPT(10, rV_CH2/10*LOG(cMaxPressure/cMinPressure) + LOG(cMinPressure))); //manual page 70 IM540 (Mode Full), (Scale) = Log

(*Pressure gauge State checks*)
//CH1
IF NOT i_xCH2_SEL AND IG_CH1.xHV_SW THEN
    IF NOT i_xERR_CH1 THEN
        IG_CH1.eState := GaugeDisconnected;
        IG_CH1.rPRESS := 0;
    ELSIF rV_CH1 <= cGaugeMaxVoltage AND rV_CH1 >= cGaugeMinVoltage AND IG_CH1.i_xHV_ON THEN
        IG_CH1.eState := Valid; // NORMAL
    ELSIF rV_CH1 >= 0.0 AND rV_CH1 < cGaugeMinVoltage AND IG_CH1.i_xHV_ON THEN
        IG_CH1.eState := OoR; //Out of range according to manual
    ELSIF rV_CH1 > cGaugeMaxVoltage AND rV_CH1 < (cGaugeMaxVoltage + cDeadband) AND IG_CH1.i_xHV_ON THEN
        IG_CH1.eState := OoR; //Out of range according to manual
    ELSIF rV_CH1 > (cGaugeMaxVoltage + cDeadband) AND tHvDis_CH1.Q THEN
        IG_CH1.eState := GaugeDisconnected; //gauge disconnected
        IG_CH1.rPRESS := 0;
    ELSIF rV_CH1 > (cGaugeMaxVoltage + cDeadband) AND NOT tHvDis_CH1.Q THEN
        IG_CH1.eState := Starting; //gauge is starting
        IG_CH1.rPRESS := 0;
    ELSE
        IG_CH1.eState := PressInvalid; //other fault - could be no gauge, controller powering up etc.
        IG_CH1.rPRESS := 0;
    END_IF
ELSE
    IG_CH1.eState := Off; // Gauge turned OFF
    IG_CH1.rPRESS := 0;
END_IF

//CH2
IF i_xCH2_SEL AND IG_CH2.xHV_SW THEN
    IF NOT i_xERR_CH2 THEN
        IG_CH2.eState := GaugeDisconnected;
        IG_CH2.rPRESS := 0;
    ELSIF rV_CH2 <= cGaugeMaxVoltage AND rV_CH2 >= cGaugeMinVoltage AND IG_CH2.i_xHV_ON THEN
        IG_CH2.eState := Valid; // NORMAL
    ELSIF rV_CH2 >= 0.0 AND rV_CH2 < cGaugeMinVoltage AND IG_CH2.i_xHV_ON THEN
        IG_CH2.eState := OoR; //Out of range according to manual
    ELSIF rV_CH2 > cGaugeMaxVoltage AND rV_CH2 < (cGaugeMaxVoltage + cDeadband) AND IG_CH2.i_xHV_ON THEN
        IG_CH2.eState := OoR; //Out of range according to manual
    ELSIF rV_CH2 > (cGaugeMaxVoltage + cDeadband) AND tHvDis_CH2.Q THEN
        IG_CH2.eState := GaugeDisconnected; //gauge disconnected
        IG_CH2.rPRESS := 0;
    ELSIF rV_CH2 > (cGaugeMaxVoltage + cDeadband) AND NOT tHvDis_CH2.Q THEN
        IG_CH2.eState := Starting; //gauge is starting
        IG_CH2.rPRESS := 0;
    ELSE
        IG_CH2.eState := PressInvalid; //other fault - could be no gauge, controller powering up etc.
        IG_CH2.rPRESS := 0;
    END_IF
ELSE
    IG_CH2.eState := Off; // Gauge turned OFF
    IG_CH2.rPRESS := 0;
END_IF

(* Ion Gauge Protection Functions *)
(* If the PG pressure is greater than the VG.PRO_SP then the gauge is disabled *)
(* If the PG pressure is less than the VG.PRO_SP then the gauge is enabled *)
(* This FB also implements some hysteresis so the gauge doesn't have rapid power cycling while near the turn on boundary *)

//CH1
IF (PG.rPRESS <= IG_CH1.rPRO_SP) AND PG.xPRESS_OK THEN
    IG_CH1.q_xHV_DIS := IG_CH1.xHV_SW;
    IG_CH1.xILKOk := TRUE;
ELSIF IG_CH1.q_xHV_DIS AND tHvDis_CH1.Q THEN
    IF IG_CH1.rPRESS > (IG_CH1.rPRO_SP + IG_CH1.rHYS_PR) OR PG.rPRESS > (IG_CH1.rPRO_SP + IG_CH1.rHYS_PR) THEN
        IG_CH1.q_xHV_DIS := FALSE;
        IG_CH1.xHV_SW := FALSE;
    END_IF
    //Adding this line because in case of interlocking gauge with another GCC or GHC PG.rPRESS value become 0 when turning it off
    IF PG.rPRESS = 0 AND NOT PG.xPRESS_OK THEN
        IG_CH1.q_xHV_DIS := FALSE;
        IG_CH1.xHV_SW := FALSE;
    END_IF
ELSE
    IG_CH1.q_xHV_DIS := FALSE;
    IG_CH1.xHV_SW := FALSE;
    IG_CH1.xILKOk := FALSE;
END_IF

//CH2
IF (PG.rPRESS <= IG_CH2.rPRO_SP) AND PG.xPRESS_OK THEN
    IG_CH2.q_xHV_DIS := IG_CH2.xHV_SW;
    IG_CH2.xILKOk := TRUE;
ELSIF IG_CH2.q_xHV_DIS AND tHvDis_CH2.Q THEN
    IF IG_CH2.rPRESS > (IG_CH2.rPRO_SP + IG_CH2.rHYS_PR) OR PG.rPRESS > (IG_CH2.rPRO_SP + IG_CH2.rHYS_PR) THEN
        IG_CH2.q_xHV_DIS := FALSE;
        IG_CH2.xHV_SW := FALSE;
    END_IF
    //Adding this line because in case of interlocking gauge with another GCC or GHC PG.rPRESS value become 0 when turning it off
    IF PG.rPRESS = 0 AND NOT PG.xPRESS_OK THEN
        IG_CH2.q_xHV_DIS := FALSE;
        IG_CH2.xHV_SW := FALSE;
    END_IF
ELSE
    IG_CH2.q_xHV_DIS := FALSE;
    IG_CH2.xHV_SW := FALSE;
    IG_CH2.xILKOk := FALSE;
END_IF


(*Pressure gauge OK checks, Backwards compatibility*)
IG_CH1.xPRESS_OK := ((IG_CH1.eState = Valid) OR IG_CH1.xBAKEOUT);
IG_CH2.xPRESS_OK := ((IG_CH2.eState = Valid) OR IG_CH2.xBAKEOUT);

(*Setpoint evaluation*)
IG_CH1.xAT_VAC := IG_CH1.xPRESS_OK AND IG_CH1.rPRESS < IG_CH1.rVAC_SP;
IG_CH2.xAT_VAC := IG_CH2.xPRESS_OK AND IG_CH2.rPRESS < IG_CH2.rVAC_SP;

(*Logger*)
ACT_Logger();

(*Soft IO Linking*)
IO();

(*Load or save the persistent variables*)
ACT_Persistent();

ACTION ACT_Logger:
// ILK logger
(*CH1 of IM540 Controller*)
IF (IG_CH1.xLog) THEN
    IF NOT IG_CH1.xILKOk AND IG_CH1.q_xHV_DIS THEN
            fbLogger(sMsg:='Lost external interlock while gauge(CH1) was on.', eSevr:=TcEventSeverity.Critical);
    END_IF

    // Log Action
    tAction_CH1(CLK := IG_CH1.xHV_SW);
    IF tAction_CH1.Q THEN fbLogger(sMsg:='Ion gauge(CH1) commanded to switch on', eSevr:=TcEventSeverity.Info); END_IF

    //STATE Logger
    IF ePrevStateIG_CH1 <> IG_CH1.eState THEN
          CASE IG_CH1.eState OF
            ValidHi:
                fbLogger(sMsg:='Gauge(CH1) pressure valid high.', eSevr:=TcEventSeverity.Info);
            ValidLo:
                fbLogger(sMsg:='Gauge(CH1) pressure valid low.', eSevr:=TcEventSeverity.Info);
            Valid:
                fbLogger(sMsg:='Gauge(CH1) pressure valid.', eSevr:=TcEventSeverity.Info);
            GaugeDisconnected:
                fbLogger(sMsg:='Gauge(CH1) Disconnected.', eSevr:=TcEventSeverity.Critical);
            PressInvalid:
                fbLogger(sMsg:='Gauge(CH1) pressure invalid.', eSevr:=TcEventSeverity.Warning);
            OoR:
                fbLogger(sMsg:='Gauge(CH1) pressure out of range.', eSevr:=TcEventSeverity.Warning);
            Starting:
                fbLogger(sMsg:='Gauge(CH1) starting.', eSevr:=TcEventSeverity.Info);
          END_CASE
          ePrevStateIG_CH1 := IG_CH1.eState;
      END_IF
END_IF

(*CH2 of IM540 Controller*)
IF (IG_CH2.xLog) THEN
    IF NOT IG_CH2.xILKOk AND IG_CH2.q_xHV_DIS THEN
            fbLogger(sMsg:='Lost external interlock while gauge(CH2) was on.', eSevr:=TcEventSeverity.Critical);
    END_IF

    // Log Action
    tAction_CH2(CLK := IG_CH2.xHV_SW);
    IF tAction_CH2.Q THEN fbLogger(sMsg:='Ion gauge(CH2) commanded to switch on', eSevr:=TcEventSeverity.Info); END_IF

    //STATE Logger
    IF ePrevStateIG_CH2 <> IG_CH2.eState THEN
          CASE IG_CH2.eState OF
            ValidHi:
                fbLogger(sMsg:='Gauge(CH2) pressure valid high.', eSevr:=TcEventSeverity.Info);
            ValidLo:
                fbLogger(sMsg:='Gauge(CH2) pressure valid low.', eSevr:=TcEventSeverity.Info);
            Valid:
                fbLogger(sMsg:='Gauge(CH2) pressure valid.', eSevr:=TcEventSeverity.Info);
            GaugeDisconnected:
                fbLogger(sMsg:='Gauge(CH2) Disconnected.', eSevr:=TcEventSeverity.Critical);
            PressInvalid:
                fbLogger(sMsg:='Gauge(CH2) pressure invalid.', eSevr:=TcEventSeverity.Warning);
            OoR:
                fbLogger(sMsg:='Gauge(CH2) pressure out of range.', eSevr:=TcEventSeverity.Warning);
            Starting:
                fbLogger(sMsg:='Gauge(CH2) starting.', eSevr:=TcEventSeverity.Info);
          END_CASE
          ePrevStateIG_CH2 := IG_CH2.eState;
      END_IF
END_IF
END_ACTION

ACTION ACT_Persistent:
(*On first PLC pass, load the persistent value into the structrue variable*)
IF (SUPER^.bRestorePersistentData) THEN
    SUPER^.bRestorePersistentData := FALSE;
    //CH1
    IF (rVAC_SP_CH1 <> 0) THEN
        IG_CH1.rVAC_SP := rVAC_SP_CH1;
    END_IF;
    IF (rPRO_SP_CH1 <> 0) THEN
        IG_CH1.rPRO_SP := rPRO_SP_CH1;
    END_IF;
    IF (rHYS_PR_CH1 <> 0) THEN
        IG_CH1.rHYS_PR := rHYS_PR_CH1;
    END_IF;
    //CH2
    IF (rVAC_SP_CH2 <> 0) THEN
        IG_CH2.rVAC_SP := rVAC_SP_CH2;
    END_IF;
    IF (rPRO_SP_CH2 <> 0) THEN
        IG_CH2.rPRO_SP := rPRO_SP_CH2;
    END_IF;
    IF (rHYS_PR_CH2 <> 0) THEN
        IG_CH2.rHYS_PR := rHYS_PR_CH2;
    END_IF;
END_IF
(*Check if a new value has been written in the structure variable copy it to the persistent variable*)
//CH1
IF NOT (IG_CH1.rVAC_SP = rVAC_SP_CH1)  THEN
    rVAC_SP_CH1 := IG_CH1.rVAC_SP;
END_IF;

IF NOT (IG_CH1.rPRO_SP = rPRO_SP_CH1) THEN
    rPRO_SP_CH1 := IG_CH1.rPRO_SP;
END_IF;

IF NOT (IG_CH1.rHYS_PR = rHYS_PR_CH1) THEN
    rHYS_PR_CH1 := IG_CH1.rHYS_PR;
END_IF;

//CH2
IF NOT (IG_CH2.rVAC_SP = rVAC_SP_CH2)  THEN
    rVAC_SP_CH2 := IG_CH2.rVAC_SP;
END_IF;

IF NOT (IG_CH2.rPRO_SP = rPRO_SP_CH2) THEN
    rPRO_SP_CH2 := IG_CH2.rPRO_SP;
END_IF;

IF NOT (IG_CH2.rHYS_PR = rHYS_PR_CH2) THEN
    rHYS_PR_CH2 := IG_CH2.rHYS_PR;
END_IF;
END_ACTION

ACTION IO:
(*soft link inputs*)
IF NOT i_xCH2_SEL THEN
    IG_CH1.i_xHV_ON := i_xHV_ON;
    IG_CH2.i_xHV_ON := FALSE;
ELSE
    IG_CH1.i_xHV_ON := FALSE;
    IG_CH2.i_xHV_ON := i_xHV_ON;
END_IF

IG_CH1.i_iPRESS_R := i_iPRESS_R_CH1;
IG_CH2.i_iPRESS_R := i_iPRESS_R_CH2;

(*soft link outputs*)
q_xHV_DIS_CH1 := IG_CH1.q_xHV_DIS;
q_xHV_DIS_CH2 := IG_CH2.q_xHV_DIS;

IG_CH1.sPath := sPath;
IG_CH2.sPath := sPath;
END_ACTION

METHOD M_AutoOnCh1 : BOOL
VAR_INPUT
END_VAR
this^.IG_CH1.q_xHV_DIS := TRUE;
END_METHOD

METHOD M_AutoOnCh2 : BOOL
VAR_INPUT
END_VAR
this^.IG_CH2.q_xHV_DIS := TRUE;
END_METHOD

METHOD M_HVECh1 : BOOL
VAR_INPUT
        enable : BOOL; // set to true to enable, false to disable;
END_VAR
this^.IG_CH1.xHV_SW := (enable);
END_METHOD

METHOD M_HVECh2 : BOOL
VAR_INPUT
        enable : BOOL; // set to true to enable, false to disable;
END_VAR
this^.IG_CH2.xHV_SW := (enable);
END_METHOD

METHOD M_IsCh1Selected : BOOL
VAR_INPUT
END_VAR
M_IsCh1Selected := NOT i_xCH2_SEL;
END_METHOD

METHOD M_IsCh2Selected : BOOL
VAR_INPUT
END_VAR
M_IsCh2Selected := i_xCH2_SEL;
END_METHOD

METHOD M_SetBits
VAR_INPUT
    TermBits : UINT; // The beckhoff terminal's maximum value in bits
END_VAR
this^.iTermBits := TermBits;
END_METHOD

END_FUNCTION_BLOCK

// ---- POUs/Functions/Gauges/FB_MX7M.TcPOU
(* This function is for the Cold Cathode MX7M from Televac. *)
(*This function provides ILK and Set Point Protection for the Cold Cathode*)
FUNCTION_BLOCK FB_MX7M EXTENDS FB_GaugeBase
VAR_IN_OUT

END_VAR
VAR_INPUT
    PG : ST_VG;
    tRecoverDelay : TIME := T#600S; (*Delay Time after the first cycle to start the device. Default is 600S*)
END_VAR
VAR_OUTPUT
    {attribute 'pytmc' := '
    pv:
    '}
    IG : ST_VG;
END_VAR
VAR
    rV : REAL; //Calculated raw voltage from ADC on analog input
    rPress : REAL; //Calculated pressure
    tGaugeTurnOnTmr : TON;
    iTermBits : UINT := 30518 ; //The terminal's maximum value in bits

    (*IOs to be linked*)
    //Controls and I/Os
    i_iPRESS_R AT %I* : INT; //Pressure reading // 'TcLinkTo' (EL3174-0002 or EP3174-0002)^Input
    q_xHV_DIS AT %Q* : BOOL; //Enable High Voltage when True // 'TcLinkTo' (EL2624 or EP2624-0002)^Output
END_VAR
VAR CONSTANT
    //Ranges 1.0 to 10.0 Vdc (1E-11 to 1E-2) 1.0V to ~1.7V indicates that the pressure is lower than 5E-11(lowest value)
    //Must set the analog output scaling to logaritmic 2!!
    cSlope : REAL := 1.0;
    cBaseV : REAL := 1.0;
    cBaseP : REAL := 1E-11;
    cMinP : REAL := 5E-11;
    cGaugeMinV : REAL := 1.0;
    cGaugeLowV : REAL := 1.69;
    cGaugeMaxV : REAL := 10.0;
    cGaugeStartingV : REAL := 10.5;
    cDefaultP : REAL := 0.0;
    cDeadbandV : REAL := 0.1;
END_VAR
VAR PERSISTENT
    bWasOn : BOOL;
    bAutoRecover : BOOL;
    bAutoRecoverWrite : BOOL;
END_VAR

(*Calculate raw voltage*)
IF (iTermBits = 0) THEN iTermBits := 30518; END_IF
rV := 10*INT_TO_REAL(i_iPRESS_R)/iTermBits;

(*Calculate pressure*)
rPRESS := LREAL_TO_REAL(EXPT(10,((rV-cBaseV)/cSlope+LOG(cBaseP))));

(*Set Guage State based on the Analog voltage*)
IF IG.q_xHV_DIS THEN
    IF rV >= cGaugeLowV AND rV < cGaugeMaxV THEN
        IG.eState := Valid;
        IG.rPRESS := rPRESS;
    ELSIF rV < cGaugeLowV AND rV >= cGaugeMinV - cDeadbandV THEN
        IG.eState := Valid;
        IG.rPRESS := cMinP;
    ELSIF rV > cGaugeStartingV - cDeadbandV THEN
        IG.eState := Starting;
        IG.rPRESS := cDefaultP;
    ELSIF rV < cGaugeMinV - cDeadbandV THEN
        IG.eState := GaugeDisconnected;
        IG.rPRESS := cDefaultP;
    ELSIF rV > cGaugeMaxV AND rV < cGaugeStartingV - cDeadbandV THEN
        IG.eState := OoR;
        IG.rPRESS := cDefaultP;
    ELSIF rV = cGaugeMaxV THEN
        IG.eState := Off;
        IG.rPRESS := cDefaultP;
    ELSE
        IG.eState := PressInvalid;
        IG.rPRESS := cDefaultP;
    END_IF
ELSE
    IG.eState := Off;
    IG.rPRESS := cDefaultP;
END_IF


(* Ion Gauge Protection Functions *)
(* If the PG pressure is greater than the VG.PRO_SP then the gauge is disabled *)
(* If the PG pressure is less than the VG.PRO_SP then the gauge is enabled *)
(* This FB also implements some hysteresis so the gauge doesn't have rapid power cycling while near the turn on boundary *)
IF PG.rPRESS <= IG.rPRO_SP AND PG.xPRESS_OK THEN
    IG.q_xHV_DIS := IG.xHV_SW;
    IG.xILKOk := TRUE;
ELSIF IG.q_xHV_DIS THEN
    IF IG.rPRESS > (IG.rPRO_SP + IG.rHYS_PR)  OR PG.rPRESS > (IG.rPRO_SP + IG.rHYS_PR) THEN
        IG.q_xHV_DIS := FALSE;
        IG.xHV_SW := FALSE;
    END_IF
ELSE
    IG.q_xHV_DIS := FALSE;
    IG.xHV_SW := FALSE;
    IG.xILKOk := FALSE;
END_IF


(*Pressure gauge OK checks*)
tGaugeTurnOnTmr(IN:=IG.q_xHV_DIS, PT:=T#10S, Q=>IG.xTurnOnTime);

//Backwards compatibility
IG.xPRESS_OK := (IG.eState = Valid) OR IG.xBAKEOUT;

(*Setpoint evaluation*)
IG.xAT_VAC := (IG.xPRESS_OK AND (IG.rPRESS < IG.rVAC_SP)) OR IG.xBAKEOUT AND (IG.eState = Valid);

(*Logging*)
ACT_Logger();

(*Soft IO Linking*)
IO();

(*Load or save the persistent variables*)
ACT_Persistent();

(*Run Auto Recovery*)
ACT_Recover();

ACTION ACT_Logger:
// ILK logger
IF (IG.xLog) THEN
    IF NOT IG.xILKOk AND IG.q_xHV_DIS THEN
            fbLogger(sMsg:='Lost external interlock while gauge was on.', eSevr:=TcEventSeverity.Critical);
    END_IF


    // Log Action
    tAction(CLK := IG.xHV_SW);
    IF tAction.Q THEN fbLogger(sMsg:='Ion gauge commanded to switch on', eSevr:=TcEventSeverity.Info); END_IF



    //STATE Logger
    IF ePrevState <> IG.eState THEN
          CASE IG.eState OF
            ValidHi:
                fbLogger(sMsg:='Gauge pressure valid high.', eSevr:=TcEventSeverity.Info);
            ValidLo:
                fbLogger(sMsg:='Gauge pressure valid low.', eSevr:=TcEventSeverity.Info);
            Valid:
                fbLogger(sMsg:='Gauge pressure valid.', eSevr:=TcEventSeverity.Info);
            GaugeDisconnected:
                fbLogger(sMsg:='Gauge Disconnected.', eSevr:=TcEventSeverity.Critical);
            PressInvalid:
                fbLogger(sMsg:='Gauge pressure invalid.', eSevr:=TcEventSeverity.Warning);
            OoR:
                fbLogger(sMsg:='Gauge pressure out of range.', eSevr:=TcEventSeverity.Warning);
            Starting:
                fbLogger(sMsg:='Gauge starting.', eSevr:=TcEventSeverity.Info);
          END_CASE
      ePrevState := IG.eState;
      END_IF
END_IF
END_ACTION

ACTION ACT_Persistent:
(*On first PLC pass, load the persistent value into the structrue variable*)
IF (SUPER^.bRestorePersistentData) THEN
    SUPER^.bRestorePersistentData := FALSE;
    IF (rVAC_SP <> 0) THEN
        IG.rVAC_SP := rVAC_SP;
    END_IF;
    IF (rPRO_SP <> 0) THEN
        IG.rPRO_SP := rPRO_SP;
    END_IF;
    IF (rHYS_PR <> 0) THEN
        IG.rHYS_PR := rHYS_PR;
    END_IF;
    IF (bAutoRecoverWrite) THEN
        IG.xAutoOn := bAutoRecover;
    END_IF;
END_IF
(*Check if a new value has been written in the structure variable copy it to the persistent variable*)
IF NOT (IG.rVAC_SP = rVAC_SP)  THEN
    rVAC_SP := IG.rVAC_SP;
END_IF;

IF NOT (IG.rPRO_SP = rPRO_SP) THEN
    rPRO_SP := IG.rPRO_SP;
END_IF;

IF NOT (IG.rHYS_PR = rHYS_PR) THEN
    rHYS_PR := IG.rHYS_PR;
END_IF;

IF NOT(bAutoRecoverWrite) OR NOT (bAutoRecover = IG.xAutoOn) THEN
    bAutoRecover := IG.xAutoOn;
    bAutoRecoverWrite := TRUE;
END_IF;

stateTimer(PT := T#10S);
IF (stateTimer.Q) THEN
    bWasOn := (IG.eState >= Valid);
    stateTimer.IN := FALSE;
    fbWritePersistentData(NETID:='', PORT:=851, START:=TRUE, TMOUT:=T#1s);
END_IF;
END_ACTION

ACTION ACT_Recover:
fbGetCurTaskIdx();
IF (TwinCAT_SystemInfoVarList._TaskInfo[fbGetCurTaskIdx.index].FirstCycle) THEN
    tRecover.IN := TRUE;
END_IF
tRecover(PT := tRecoverDelay);
IF NOT(bAutoRecoverWrite) OR (tRecover.Q AND bAutoRecover) THEN
    This^.M_Recover();
    tRecover.IN := FALSE;
END_IF
END_ACTION

ACTION IO:
(*soft link inputs*)
IG.i_iPRESS_R := i_iPRESS_R;
IG.i_xHV_ON := IG.q_xHV_DIS;  //not a real readback, assuming turning on HV output, HV status is ON and vice versa

(*soft link outputs*)
q_xHV_DIS := IG.q_xHV_DIS;

(*Gauge name link*)
IG.sPath := sPath;
END_ACTION

METHOD M_HVE : BOOL
VAR_INPUT
        bEnable : BOOL; // set to true to enable, false to disable;
END_VAR
this^.IG.xHV_SW := bEnable;
END_METHOD

METHOD M_Recover : BOOL
VAR_INPUT
END_VAR
This^.M_HVE(This^.bWasOn);
M_Recover := bWasOn;
IF (bWasOn) THEN fbLogger(sMsg:='Auto Recovery Initiated.', eSevr:=TcEventSeverity.Info); END_IF;
END_METHOD

METHOD M_SetBits : BOOL
VAR_INPUT
    TermBits : UINT; // The terminal's maximum value in bits
END_VAR
This^.iTermBits := TermBits;
END_METHOD

END_FUNCTION_BLOCK

// ---- POUs/Functions/Gauges/FB_CVM201.TcPOU
(* This function block is used to provide protection and automatic turn on of ion gauges,
 it also manages the turn on of the AT_VAC boolean, and checks to make sure the pressure is good *)
(* For CVM 201  convectron SuperBee*)
{attribute 'no_check'}
FUNCTION_BLOCK FB_CVM201 EXTENDS FB_GaugeBase
VAR_IN_OUT

END_VAR
VAR_INPUT
END_VAR

VAR_OUTPUT
    {attribute 'pytmc' := '
    pv:
    '}
    PG : ST_VG;
END_VAR
VAR
    V : REAL;
    iTermBits: UINT := 32767 ; // The terminal's maximum value in bits
    Vlowest: REAL := 10;
    (*IO*)
    i_iPRESS_R AT%I* :INT; // input Pressure // Link to analog Input
END_VAR

VAR CONSTANT
    MinPressure: REAL := 1E-4;
    rDeadband : REAL :=0.05;
    rValidLoBoundary	:	REAL := 0.375; //  0.375V as per manual page 27
    rValidHiBoundary	:	REAL := 5.659;// 5.534; // manual page 27
    rDisconnectedBoundary	:	REAL := 0.3;
    (*Default set point 50 mT*)
    rDefaultVAC_SP: REAL := 5E-2;
END_VAR

(* This function block is used to provide protection and automatic turn on of ion gauges,
 it also manages the turn on of the AT_VAC boolean, and checks to make sure the pressure is good *)
(* For MKS 275 mini-convectron *)

//Default setpoint 50 mT
IF PG.rVAC_SP = 0 THEN
    PG.rVAC_SP := 5E-2;
END_IF

(* Real-value calculation *)
If (iTermBits=0) THEN iTermBits := 32767;END_IF
V := 10*INT_TO_REAL(PG.i_iPRESS_R)/iTermBits;

Vlowest := MIN(V, Vlowest);

IF V > rDisconnectedBoundary AND V < rValidLoBoundary  THEN
    PG.rPRESS := MinPressure;
    PG.eState := ValidLo;

ELSIF V >= rValidLoBoundary AND V < rValidLoBoundary +rDeadband  THEN
    PG.rPRESS := MAX( MinPressure, LREAL_TO_REAL( -0.02585 + 0.03767*V + 0.04563*EXPT(V,2)+ 0.1151*EXPT(V,3) - 0.04158*EXPT(V,4)+ 0.008737*EXPT(V,5)) );
    PG.eState := ValidLo;

ELSIF V >= rValidLoBoundary AND V < 2.842 THEN
    PG.rPRESS := MAX( MinPressure, LREAL_TO_REAL( -0.02585 + 0.03767*V + 0.04563*EXPT(V,2)+ 0.1151*EXPT(V,3) - 0.04158*EXPT(V,4)+ 0.008737*EXPT(V,5)) );
    PG.eState := Valid;

ELSIF V >= 2.842 AND V < 4.945 THEN
    PG.rPRESS := LREAL_TO_REAL((0.1031-0.02322*V+0.07229*EXPT(V,2))/(1-0.3986*V+0.07438*EXPT(V,2)-0.006866*EXPT(V,3)));
    PG.eState := Valid;

ELSIF V >= 4.945 AND V < rValidHiBoundary THEN
    PG.rPRESS := LREAL_TO_REAL((100.624-20.5623*V)/(1-0.37679*V+0.0348656*EXPT(V,2)));
    PG.eState := ValidHi;

ELSIF V <= rDisconnectedBoundary THEN
    PG.eState := GaugeDisconnected; //Most likely not connected
    PG.rPRESS := -1;

ELSE
    PG.eState := OoR; //Larger voltage, probably out of range?
    PG.rPRESS := -1;
END_IF

(* Protection Functions *)
(* If the PG pressure is greater than the IG.PRO_SP then the gauge is disabled *)
(* If the PG pressure is less than the IG.PRO_SP then the gauge is enabled *)
(* This FB also implements some hysteresis so the gauge doesn't have rapid power cycling while near the turn on boundary *)

(* Pressure OK check *)
PG.xPRESS_OK := (PG.rPRESS >= MinPressure);

(* Setpoint evaluation *)
PG.xAT_VAC := PG.xPRESS_OK AND (PG.rPRESS<=PG.rVAC_SP);

(*Logger*)
ACT_Logger();

(*Soft IO Mapping *)
IO();

(*Load or save the persistent variables*)
ACT_Persistent();

ACTION ACT_Logger:

//STATE Logger
if (PG.xLog) THEN
    IF ePrevState <> PG.eState THEN
      CASE PG.eState OF
        ValidHi:
            fbLogger(sMsg:='Gauge pressure valid high.', eSevr:=TcEventSeverity.Info);
        ValidLo:
            fbLogger(sMsg:='Gauge pressure valid low.', eSevr:=TcEventSeverity.Info);
        Valid:
            fbLogger(sMsg:='Gauge pressure valid.', eSevr:=TcEventSeverity.Info);
          GaugeDisconnected:
            fbLogger(sMsg:='Gauge Disconnected.', eSevr:=TcEventSeverity.Critical);
        PressInvalid:
            fbLogger(sMsg:='Gauge pressure invalid.', eSevr:=TcEventSeverity.Warning);
        OoR:
            fbLogger(sMsg:='Gauge pressure out of range.', eSevr:=TcEventSeverity.Warning);
        Starting:
            fbLogger(sMsg:='Gauge starting.', eSevr:=TcEventSeverity.Info);
      END_CASE
      ePrevState := PG.eState;
  END_IF
END_IF
END_ACTION

ACTION ACT_Persistent:
(*On first PLC pass, load the persistent value into the structrue variable*)
IF (SUPER^.bRestorePersistentData) THEN
    SUPER^.bRestorePersistentData	:= FALSE;
    IF (rPRO_SP <> 0) THEN
        PG.rPRO_SP := rPRO_SP;
    END_IF;
END_IF
(*Check if a new value has been written in the structure variable copy it to the persistent variable*)
IF NOT (PG.rVAC_SP = rVAC_SP) THEN
    rVAC_SP:= PG.rVAC_SP;
END_IF;
END_ACTION

ACTION IO:
PG.i_iPRESS_R :=i_iPRESS_R;
PG.sPath := sPath;
END_ACTION

METHOD M_SetBits : BOOL
VAR_INPUT
    TermBits : UINT; // The terminal's maximum value in bits
END_VAR
This^.iTermBits := TermBits;
END_METHOD

END_FUNCTION_BLOCK

// ---- POUs/Functions/Gauges/FB_CCM501.TcPOU
(* This function is for the Cold Cathode CCM 501 fro instrutech (hornet). *)
(*This function provides ILK and Set Point Protection for the Cold Cathode*)

FUNCTION_BLOCK FB_CCM501 EXTENDS FB_GaugeBase
VAR_IN_OUT

END_VAR
VAR_INPUT
    PG	:	ST_VG;
//	bEP : BOOL :=FALSE; // Set to True if This Gauge is connected to EP BOX and not EL Terminals
    tRecoverDelay:TIME:=T#600S; (*Delay Time after the first cycle to start the device. Default is 600S*)
END_VAR
VAR_OUTPUT
{attribute 'pytmc' := '
    pv:
    '}
    IG : ST_VG;
END_VAR
VAR
    rV : REAL;
    GaugeTurnOnTmr : TON;
    tStartupTimer:TON;
    iTermBits: UINT := 30518 ; // The terminal's maximum value in bits
    (*IOs to be linked*)
    /// Controls and I/Os
    i_iPRESS_R AT %I* :INT; // input Pressure // Link to analog Input
    q_xHV_DIS AT %Q* : BOOL; // Enable High Voltage when True // 'TcLinkTo' (EP2624) ^Output
    // only for EL and ES terminal
    i_xHV_ON AT %I*	: BOOL; //  True when High Voltage is on  // 'TcLinkTo' (EL1124) ^Input
//	i_xDisc_Active AT %I* : BOOL;// Discharge Current Active // 'TcLinkTo' (EL1124) ^Input
    binit:BOOL:=TRUE;
END_VAR

VAR CONSTANT
    // Ranges 1.8 to 8.7 Vdc, 0.8V/decade analog output - Torr
    vBase : REAL := 1.25;
    vDisconnected : REAL:= 1.8;
    vTorr : REAL := 12.875;
    vGaugeOff: REAL := 10.0;
    //vNoDischarge: REAL := 9.3;
    rMinPressure: REAL := 1E-10;
    cDefaultPressure : REAL := 0;
    rDeadband : REAL := 1.0;
END_VAR
VAR PERSISTENT
    bWasOn : BOOL;
    bAutoRecover:BOOL;
    bAutoRecoverWrite:BOOL;
END_VAR


(*Startup time*)
IF (bInit) THEN
    tStartupTimer.IN:=TRUE;
    bInit :=FALSE;
END_IF
tStartupTimer(PT:=T#3S);



If (iTermBits=0) THEN iTermBits := 30518;END_IF
rV := 10*INT_TO_REAL(IG.i_iPRESS_R)/iTermBits;

(* Set Guage State based on the Analog voltage*)
IF rV <= vDisconnected AND IG.i_xHV_ON AND IG.q_xHV_DIS THEN
    IG.eState := ValidLo;
    IG.rPRESS := rMinPressure;
ELSIF rV <= vDisconnected AND NOT IG.i_xHV_ON AND IG.q_xHV_DIS THEN
    IG.eState := GaugeDisconnected;
    IG.rPRESS := cDefaultPressure;
ELSIF rV > vDisconnected AND rV < (vGaugeOff -rDeadband) AND IG.i_xHV_ON AND IG.q_xHV_DIS THEN
    IG.eState := Valid;
    IG.rPRESS := LREAL_TO_REAL(EXPT(10,((rV*vBase)- vTorr)));
ELSIF rV >= (vGaugeOff -rDeadband) AND IG.i_xHV_ON AND IG.q_xHV_DIS THEN
    IG.eState := Starting;
    IG.rPRESS := cDefaultPressure;
ELSIF rV >= (vGaugeOff -rDeadband) THEN
    IG.eState := Off;
    IG.rPRESS := cDefaultPressure;
ELSE
    IG.eState := OoR;
    IG.rPRESS := cDefaultPressure;
END_IF




(* Ion Gauge Protection Functions *)
(* If the PG pressure is greater than the VG.PRO_SP then the gauge is disabled *)
(* If the PG pressure is less than the VG.PRO_SP then the gauge is enabled *)
(* This FB also implements some hysteresis so the gauge doesn't have rapid power cycling while near the turn on boundary *)


IF PG.rPRESS <= IG.rPRO_SP AND PG.xPRESS_OK THEN
    IG.q_xHV_DIS := IG.xHV_SW;
    IG.xILKOk := TRUE;
ELSIF IG.q_xHV_DIS THEN
    IF IG.rPRESS > (IG.rPRO_SP + IG.rHYS_PR)  OR PG.rPRESS > (IG.rPRO_SP + IG.rHYS_PR) THEN
        IG.q_xHV_DIS := FALSE;
        IG.xHV_SW := FALSE;
    END_IF
ELSE
    IG.q_xHV_DIS := FALSE;
    IG.xHV_SW := FALSE;
    IG.xILKOk := FALSE;
END_IF


(* Pressure gauge OK checks *)
GaugeTurnOnTmr(IN:=IG.q_xHV_DIS, PT:=T#10S, Q=>IG.xTurnOnTime);

//Backwards compatibility
IG.xPRESS_OK := (IG.eState = Valid) OR (IG.eState = ValidLo) OR IG.xBAKEOUT;

(* Setpoint evaluation *)
IG.xAT_VAC := IG.xPRESS_OK AND (IG.rPRESS < IG.rVAC_SP);

ACT_Logger();
(*Soft IO Linking*)
// check ethercat Diagnostics
IO();
(*Load or save the persistent variables*)
ACT_Persistent();

(*Run Auto Recovery*)
ACT_Recover();

ACTION ACT_Logger:
// ILK logger
IF (IG.xLog) THEN
    IF NOT IG.xILKOk AND IG.q_xHV_DIS THEN
            fbLogger(sMsg:='Lost external interlock while gauge was on.', eSevr:=TcEventSeverity.Critical);
    END_IF


    // Log Action
    tAction(CLK:=   IG.xHV_SW);
    IF tAction.Q THEN fbLogger(sMsg:='Ion gauge commanded to switch on', eSevr:=TcEventSeverity.Info); END_IF



    //STATE Logger
    tState(CLK:=  ePrevState <> IG.eState);
    IF ePrevState <> IG.eState THEN
          CASE IG.eState OF
            ValidHi:
                fbLogger(sMsg:='Gauge pressure valid high.', eSevr:=TcEventSeverity.Info);
            ValidLo:
                fbLogger(sMsg:='Gauge pressure valid low.', eSevr:=TcEventSeverity.Info);
            Valid:
                fbLogger(sMsg:='Gauge pressure valid.', eSevr:=TcEventSeverity.Info);
            GaugeDisconnected:
                fbLogger(sMsg:='Gauge Disconnected.', eSevr:=TcEventSeverity.Critical);
            PressInvalid:
                fbLogger(sMsg:='Gauge pressure invalid.', eSevr:=TcEventSeverity.Warning);
            OoR:
                fbLogger(sMsg:='Gauge pressure out of range.', eSevr:=TcEventSeverity.Warning);
            Starting:
                fbLogger(sMsg:='Gauge starting.', eSevr:=TcEventSeverity.Info);
          END_CASE
          ePrevState := IG.eState;
      END_IF
END_IF
END_ACTION

ACTION ACT_Persistent:
(*On first PLC pass, load the persistent value into the structrue variable*)

IF (SUPER^.bRestorePersistentData) THEN
    SUPER^.bRestorePersistentData	:= FALSE;
    IF ( rVAC_SP <> 0) THEN
        IG.rVAC_SP := rVAC_SP;
    END_IF;
    IF ( rPRO_SP <> 0) THEN
        IG.rPRO_SP := rPRO_SP;
    END_IF;
    IF ( rHYS_PR <> 0) THEN
        IG.rHYS_PR := rHYS_PR;
    END_IF;
    IF ( bAutoRecoverWrite) THEN
        IG.xAutoOn := bAutoRecover;
    END_IF;
END_IF
(*Check if a new value has been written in the structure variable copy it to the persistent variable*)
IF NOT (IG.rVAC_SP = rVAC_SP)  THEN
    rVAC_SP := IG.rVAC_SP;
END_IF;

IF NOT (IG.rPRO_SP = rPRO_SP) THEN
    rPRO_SP:= IG.rPRO_SP;
END_IF;

IF NOT (IG.rHYS_PR = rHYS_PR) THEN
    rHYS_PR:= IG.rHYS_PR;
END_IF;

IF NOT(bAutoRecoverWrite) OR NOT (bAutoRecover = IG.xAutoOn) THEN
    bAutoRecover := IG.xAutoOn;
    bAutoRecoverWrite := TRUE;
END_IF;
stateTimer(PT:=T#10S);
IF (stateTimer.Q) THEN
    bWasOn := (IG.eState >=Valid );
    stateTimer.IN := FALSE;
    fbWritePersistentData(NETID:='', PORT:=851, START:=TRUE, TMOUT:=T#1s );
END_IF;
END_ACTION

ACTION ACT_Recover:
fbGetCurTaskIdx();
IF (TwinCAT_SystemInfoVarList._TaskInfo[fbGetCurTaskIdx.index].FirstCycle) THEN
    tRecover.IN := TRUE;
END_IF
tRecover(IN:= , PT:=tRecoverDelay);
IF NOT(bAutoRecoverWrite) OR (tRecover.Q AND bAutoRecover ) THEN
    This^.M_Recover();
    tRecover.IN := FALSE;
END_IF
END_ACTION

ACTION IO:
(*soft link inputs*)
IG.i_iPRESS_R:=	i_iPRESS_R;
IG.i_xHV_ON:= i_xHV_ON;
//IG.i_xDisc_Active:=i_xDisc_Active;
(*soft link outputs*)
q_xHV_DIS := IG.q_xHV_DIS;

IG.sPath := sPath;
END_ACTION

METHOD M_HVE : BOOL
VAR_INPUT
        enable:bool; // set to true to enable, false to disable;
END_VAR

this^.IG.xHV_SW:= enable;
END_METHOD

METHOD M_Recover : BOOL
VAR_INPUT
END_VAR
This^.M_HVE(This^.bWasOn);
M_Recover := bWasOn;
IF (bWasOn) THEN fbLogger(sMsg:='Auto Recovery Initiated.', eSevr:=TcEventSeverity.Info); END_IF;
END_METHOD

METHOD M_SetBits : BOOL
VAR_INPUT
    TermBits : UINT; // The terminal's maximum value in bits
END_VAR
This^.iTermBits := TermBits;
END_METHOD

END_FUNCTION_BLOCK

// ---- POUs/Functions/Gauges/FB_IMG401.TcPOU
(* This function is for the Cold Cathode MKS 500.

If connected to Beckhoff EP boxes. Set the EP bit to TRUE, this is necessary for the
IMG401-to-EP box interface because the EP boxes do not natively support the 5v IO
signals on the gauge.

This function provides ILK and Set Point Protection for the hot Cathode.
*)

FUNCTION_BLOCK FB_IMG401 EXTENDS FB_GaugeBase
VAR_IN_OUT

END_VAR
VAR_INPUT
    PG	:	ST_VG;
    tRecoverDelay:TIME:=T#600S; (*Delay Time after the first cycle to start the device. Default is 600S*)
END_VAR
VAR_OUTPUT
{attribute 'pytmc' := '
    pv:
    '}
    IG : ST_VG;
END_VAR
VAR
    rV : REAL;
    GaugeTurnOnTmr : TON;
    tStartupTimer:TON;
    iTermBits: UINT := 30518 ; // The terminal's maximum value in bits
    (*IOs to be linked*)
    /// Controls and I/Os
    i_iPRESS_R AT %I* :INT; // input Pressure // Link to analog Input
    q_xHV_DIS AT %Q* : BOOL; // Enable High Voltage when True // 'TcLinkTo' (EP2624) ^Output
    // only for EL and ES terminal
    i_xHV_ON AT %I*	: BOOL; //  True when High Voltage is on  // 'TcLinkTo' (EL1084) ^Input
//	i_xDisc_Active AT %I* : BOOL;// Discharge Current Active // 'TcLinkTo' (EL1124) ^Input
    binit:BOOL:=TRUE;
END_VAR

VAR CONSTANT
    vBase : REAL := 1.0;
    vDisconnected : REAL:= 0.001; //shift from 0 to eliminate single noise effect
    vTorr : REAL := 10;
    vGaugeOff: REAL := 10;
    //vNoDischarge: REAL := 9.3;
    rMinPressure: REAL := 1E-10;
    cDefaultPressure : REAL := 0;
    rDeadband : REAL :=1.0;
END_VAR

VAR PERSISTENT
    bWasOn : BOOL;
    bAutoRecover:BOOL;
    bAutoRecoverWrite:BOOL;
END_VAR

(*Startup time*)
IF (bInit) THEN
    tStartupTimer.IN:=TRUE;
    bInit :=FALSE;
END_IF
tStartupTimer(PT:=T#3S);

(* 401 Logarithmic Output Conversion, factory default configuration
   EL3174, EL3174-xxxx iTermbits 30518, 10V
*)
If (iTermBits=0) THEN iTermBits := 30518;END_IF
rV := 10*INT_TO_REAL(IG.i_iPRESS_R)/iTermBits;

(* Set Guage State based on the Analog voltage*)

IF rV <= vDisconnected AND IG.i_xHV_ON and IG.q_xHV_DIS THEN
    IG.eState := ValidLo;
    IG.rPRESS := rMinPressure;
ELSIF rV <= vDisconnected AND Not IG.i_xHV_ON and IG.q_xHV_DIS THEN
    IG.eState := GaugeDisconnected;
    IG.rPRESS := cDefaultPressure;
ELSIF rV > vDisconnected AND rV < (vGaugeOff -rDeadband) AND IG.i_xHV_ON and IG.q_xHV_DIS THEN
    IG.eState := Valid;
    IG.rPRESS := LREAL_TO_REAL(EXPT(10,((rV*vBase)- vTorr)));
ELSIF rV >= (vGaugeOff -rDeadband) THEN
    IG.eState := Off;
    IG.rPRESS := cDefaultPressure;
ELSE
    IG.eState := OoR;
    IG.rPRESS := cDefaultPressure;
END_IF



(* Ion Gauge Protection Functions *)
(* If the PG pressure is greater than the VG.PRO_SP then the gauge is disabled *)
(* If the PG pressure is less than the VG.PRO_SP then the gauge is enabled *)
(* This FB also implements some hysteresis so the gauge doesn't have rapid power cycling while near the turn on boundary *)


IF PG.rPRESS <= IG.rPRO_SP AND PG.xPRESS_OK THEN
    IG.q_xHV_DIS := IG.xHV_SW;
    IG.xILKOk := TRUE;
ELSIF IG.q_xHV_DIS THEN
    IF IG.rPRESS > (IG.rPRO_SP + IG.rHYS_PR)  OR PG.rPRESS > (IG.rPRO_SP + IG.rHYS_PR) THEN
        IG.q_xHV_DIS := FALSE;
        IG.xHV_SW := FALSE;
    END_IF
ELSE
    IG.q_xHV_DIS := FALSE;
    IG.xHV_SW := FALSE;
    IG.xILKOk := FALSE;
END_IF

(* Pressure gauge OK checks *)

GaugeTurnOnTmr(IN:=IG.q_xHV_DIS, PT:=T#10S, Q=>IG.xTurnOnTime);

//Backwards compatibility
IG.xPRESS_OK := (IG.eState = Valid) OR IG.xBAKEOUT;

(* Setpoint evaluation *)
IG.xAT_VAC := (IG.xPRESS_OK AND (IG.rPRESS < IG.rVAC_SP)) OR IG.xBAKEOUT AND (IG.eState = Valid) ;

ACT_Logger();
(*Soft IO Linking*)
// check ethercat Diagnostics
IO();
(*Load or save the persistent variables*)
ACT_Persistent();
(*Run Auto Recovery*)
ACT_Recover();

ACTION ACT_Logger:
// ILK logger
IF (IG.xLog) THEN
    IF NOT IG.xILKOk AND IG.q_xHV_DIS THEN
            fbLogger(sMsg:='Lost external interlock while gauge was on.', eSevr:=TcEventSeverity.Critical);
    END_IF


    // Log Action
    tAction(CLK:=   IG.xHV_SW);
    IF tAction.Q THEN fbLogger(sMsg:='Ion gauge commanded to switch on', eSevr:=TcEventSeverity.Info); END_IF



    //STATE Logger
    tState(CLK:=  ePrevState <> IG.eState);
    IF ePrevState <> IG.eState THEN
          CASE IG.eState OF
            ValidHi:
                fbLogger(sMsg:='Gauge pressure valid high.', eSevr:=TcEventSeverity.Info);
            ValidLo:
                fbLogger(sMsg:='Gauge pressure valid low.', eSevr:=TcEventSeverity.Info);
            Valid:
                fbLogger(sMsg:='Gauge pressure valid.', eSevr:=TcEventSeverity.Info);
            GaugeDisconnected:
                fbLogger(sMsg:='Gauge Disconnected.', eSevr:=TcEventSeverity.Critical);
            PressInvalid:
                fbLogger(sMsg:='Gauge pressure invalid.', eSevr:=TcEventSeverity.Warning);
            OoR:
                fbLogger(sMsg:='Gauge pressure out of range.', eSevr:=TcEventSeverity.Warning);
            Starting:
                fbLogger(sMsg:='Gauge starting.', eSevr:=TcEventSeverity.Info);
          END_CASE
          ePrevState := IG.eState;
          stateTimer.IN := TRUE;
      END_IF
END_IF
END_ACTION

ACTION ACT_Persistent:
(*On first PLC pass, load the persistent value into the structrue variable*)
IF (SUPER^.bRestorePersistentData) THEN
    SUPER^.bRestorePersistentData	:= FALSE;
    IF ( rVAC_SP <> 0) THEN
        IG.rVAC_SP := rVAC_SP;
    END_IF;
    IF ( rPRO_SP <> 0) THEN
        IG.rPRO_SP := rPRO_SP;
    END_IF;
    IF ( rHYS_PR <> 0) THEN
        IG.rHYS_PR := rHYS_PR;
    END_IF;
    IF ( bAutoRecoverWrite) THEN
        IG.xAutoOn := bAutoRecover;
    END_IF;
END_IF
(*Check if a new value has been written in the structure variable copy it to the persistent variable*)
IF NOT (IG.rVAC_SP = rVAC_SP)  THEN
    rVAC_SP := IG.rVAC_SP;
END_IF;

IF NOT (IG.rPRO_SP = rPRO_SP) THEN
    rPRO_SP:= IG.rPRO_SP;
END_IF;

IF NOT (IG.rHYS_PR = rHYS_PR) THEN
    rHYS_PR:= IG.rHYS_PR;
END_IF;

IF NOT(bAutoRecoverWrite) OR NOT (bAutoRecover = IG.xAutoOn) THEN
    bAutoRecover := IG.xAutoOn;
    bAutoRecoverWrite := TRUE;
END_IF;
stateTimer(PT:=T#10S);
IF (stateTimer.Q) THEN
    bWasOn := (IG.eState >=Valid );
    stateTimer.IN := FALSE;
    fbWritePersistentData(NETID:='', PORT:=851, START:=TRUE, TMOUT:=T#1s );
END_IF;
END_ACTION

ACTION ACT_Recover:
fbGetCurTaskIdx();
IF (TwinCAT_SystemInfoVarList._TaskInfo[fbGetCurTaskIdx.index].FirstCycle) THEN
    tRecover.IN := TRUE;
END_IF
tRecover(IN:= , PT:=tRecoverDelay);
IF NOT(bAutoRecoverWrite) OR (tRecover.Q AND bAutoRecover ) THEN
    This^.M_Recover();
    tRecover.IN := FALSE;
END_IF
END_ACTION

ACTION IO:
(*soft link inputs*)
IG.i_iPRESS_R:=	i_iPRESS_R;
IG.i_xHV_ON:= i_xHV_ON;
//IG.i_xDisc_Active:=i_xDisc_Active;
(*soft link outputs*)
q_xHV_DIS := IG.q_xHV_DIS;

IG.sPath := sPath;
IG.iAutoOnTimer:= TIME_TO_INT(tRecover.PT);
END_ACTION

METHOD M_HVE : BOOL
VAR_INPUT
        enable:bool; // set to true to enable, false to disable;
END_VAR
this^.IG.xHV_SW:= enable;
END_METHOD

METHOD M_Recover : BOOL
VAR_INPUT
END_VAR
This^.M_HVE(This^.bWasOn);
M_Recover := bWasOn;
IF (bWasOn) THEN fbLogger(sMsg:='Auto Recovery Initiated.', eSevr:=TcEventSeverity.Info); END_IF;
END_METHOD

METHOD M_SetBits : BOOL
VAR_INPUT
    TermBits : UINT; // The terminal's maximum value in bits
END_VAR
This^.iTermBits := TermBits;
END_METHOD

END_FUNCTION_BLOCK

// ---- POUs/Functions/Gauges/FB_MKS909.TcPOU
(* Standard MKS 909 hot cathode *)
(* works for 972 and 925 *)

FUNCTION_BLOCK FB_MKS909 EXTENDS FB_GaugeBase

VAR_INPUT
    PG	: ST_VG;
END_VAR
VAR_OUTPUT
    {attribute 'pytmc' := '
    pv:
    '}
    IG	: ST_VG;
END_VAR
VAR_IN_OUT

END_VAR
VAR
    rV : REAL;
    rMaxPressure	:	REAL := 5E-2; //Torr
    rMinPressure	:	REAL := 1E-10; //Torr
    timer:TON;
    (*Default set point 50 mT*)
    rDefaultVAC_SP: REAL := 9E-3; // as per manual
    iTermBits: UINT := 30518 ; // The terminal's maximum value in bits default el3174 as per vacuum architecture
    (*IO*)
    i_iPRESS_R AT%I* :INT; // input Pressure // Link to analog Input
    q_xHV_DIS AT %Q* : BOOL := TRUE; // Active Low

END_VAR

(* Standard MKS 9XX series conversion *)
(* works for 972 and 925 *)

//Default setpoint 50 mT
IF PG.rVAC_SP = 0 THEN
    PG.rVAC_SP := rDefaultVAC_SP;
END_IF
// check no div by zero
If (iTermBits=0) THEN iTermBits := 30518;END_IF
rV := 10*INT_TO_REAL(IG.i_iPRESS_R)/iTermBits;

(* Pressure OK check *)
// Gauge state
// Is the gauge plugged in, and within a reasonable range?
IF  (rV >= 0.1 AND rV <=8.7) THEN // as per manual
    IG.rPRESS := LREAL_TO_REAL(EXPT(10, rV-10));
    IG.eState := Valid;
    IG.xPRESS_OK := TRUE; //Backwards compatibility
ELSIF rV > 8.7 AND rV < 10 THEN
    IG.rPRESS :=rMaxPressure;
    IG.xPRESS_OK := FALSE;
    IG.eState := Off;
ELSE
    IG.xPRESS_OK := FALSE;
    IG.eState := GaugeDisconnected;
END_IF


IF (PG.rPRESS <= IG.rPRO_SP)  AND (PG.xPRESS_OK) THEN
         IG.q_xHV_DIS := IG.xHV_SW;
         IG.xILKOk := TRUE;
    ELSIF NOT IG.q_xHV_DIS AND timer.Q THEN
        IF IG.rPRESS > (IG.rPRO_SP + IG.rHYS_PR) OR PG.rPRESS > (IG.rPRO_SP + IG.rHYS_PR) THEN
        IG.q_xHV_DIS := FALSE;
        IG.xHV_SW := FALSE;
        END_IF
    ELSE
        IG.q_xHV_DIS := FALSE;
        IG.xHV_SW := FALSE;
        IG.xILKOk := FALSE;
     END_IF


timer(IN:= NOT IG.q_xHV_DIS, PT:= T#2s);

(* Setpoint evaluation *)
IG.xAT_VAC := IG.xPRESS_OK AND (IG.rPRESS < IG.rVAC_SP);

(*Soft IO Mapping*)
ACT_IO();
(*Load or save the persistent variables*)
ACT_Persistent();

(*Logger*)
THIS^.ACT_Logger();

(*Load or save the persistent variables*)
ACT_Persistent();

ACTION ACT_IO:
(*soft link inputs*)
IG.i_iPRESS_R:=	i_iPRESS_R;

(*soft link outputs*)
q_xHV_DIS := IG.q_xHV_DIS;
END_ACTION

ACTION ACT_Logger:
// ILK logger
IF NOT IG.xILKOk AND NOT IG.q_xHV_DIS THEN
         fbLogger(sMsg:='Lost external interlock while gauge was on.', eSevr:=TcEventSeverity.Critical);
END_IF


// Log Action
tAction(CLK:=  IG.q_xHV_DIS);
IF tAction.Q THEN fbLogger(sMsg:='Ion gauge commanded to switch on', eSevr:=TcEventSeverity.Info); END_IF



//STATE Logger
IF ePrevState <> IG.eState THEN
      CASE IG.eState OF
        ValidHi:
        ValidLo:
        Valid:
            fbLogger(sMsg:='Gauge pressure valid.', eSevr:=TcEventSeverity.Info);
          GaugeDisconnected:
            fbLogger(sMsg:='Gauge Disconnected.', eSevr:=TcEventSeverity.Critical);
        PressInvalid:
            fbLogger(sMsg:='Gauge pressure invalid.', eSevr:=TcEventSeverity.Warning);
        OoR:
            fbLogger(sMsg:='Gauge pressure out of range.', eSevr:=TcEventSeverity.Warning);
        Starting:
            fbLogger(sMsg:='Gauge starting.', eSevr:=TcEventSeverity.Info);
      END_CASE
      ePrevState := IG.eState;
END_IF
END_ACTION

ACTION ACT_Persistent:
(*On first PLC pass, load the persistent value into the structrue variable*)
IF (SUPER^.bRestorePersistentData) THEN
    SUPER^.bRestorePersistentData	:= FALSE;
    IF ( rVAC_SP <> 0) THEN
        IG.rVAC_SP := rVAC_SP;
    END_IF;
    IF ( rPRO_SP <> 0) THEN
        IG.rPRO_SP := rPRO_SP;
    END_IF;
    IF ( rHYS_PR <> 0) THEN
        IG.rHYS_PR := rHYS_PR;
    END_IF;
END_IF
(*Check if a new value has been written in the structure variable copy it to the persistent variable*)
IF NOT (IG.rVAC_SP = rVAC_SP)  THEN
    rVAC_SP := IG.rVAC_SP;
END_IF;

IF NOT (IG.rPRO_SP = rPRO_SP) THEN
    rPRO_SP:= IG.rPRO_SP;
END_IF;

IF NOT (IG.rHYS_PR = rHYS_PR) THEN
    rHYS_PR:= IG.rHYS_PR;
END_IF;
END_ACTION

METHOD M_AutoOn : BOOL
VAR_INPUT
END_VAR
this^.IG.q_xHV_DIS:= FALSE;
END_METHOD

METHOD M_SetBits : BOOL
VAR_INPUT
    TermBits : UINT; // The terminal's maximum value in bits
END_VAR
This^.iTermBits := TermBits;
END_METHOD

END_FUNCTION_BLOCK

// ---- POUs/Functions/Gauges/FB_MKS909_RBK.TcPOU
(* Standard MKS 909 hot cathode with gauge on reedback*)
(* works for 972 and 925 *)

FUNCTION_BLOCK FB_MKS909_RBK EXTENDS FB_GaugeBase

VAR_INPUT
    PG	: ST_VG;
END_VAR
VAR_OUTPUT
    {attribute 'pytmc' := '
    pv:
    '}
    IG	: ST_VG;
END_VAR
VAR_IN_OUT

END_VAR
VAR
    rV : REAL;
    rMaxPressure	:	REAL := 5E-2; //Torr
    rMinPressure	:	REAL := 1E-10; //Torr
    rOffPressure	:	REAL := 0.0;
    timer:TON;
    (*Default set point 50 mT*)
    rDefaultVAC_SP: REAL := 9E-3; // as per manual
    iTermBits: UINT := 30518 ; // The terminal's maximum value in bits default el3174 as per vacuum architecture
    (*IO*)
    i_iPRESS_R AT%I* :INT; // input Pressure // Link to analog Input
    q_xHV_DIS AT %Q* : BOOL := TRUE; // Active Low
    i_xGauge_ON AT %I*	: BOOL; //  True when gauge has power  // 'TcLinkTo' (EL1084) ^Input

END_VAR

(* Standard MKS 9XX series conversion *)
(* works for 972 and 925 *)

//Default setpoint 50 mT
IF PG.rVAC_SP = 0 THEN
    PG.rVAC_SP := rDefaultVAC_SP;
END_IF
// check no div by zero
If (iTermBits=0) THEN iTermBits := 30518;END_IF
rV := 10*INT_TO_REAL(IG.i_iPRESS_R)/iTermBits;

(* Pressure OK check *)
// Gauge state
// Is the gauge plugged in, and within a reasonable range?
IF i_xGauge_ON THEN
    IF  (rV >= 0.1 AND rV <=8.7) THEN // as per manual
        IG.rPRESS := LREAL_TO_REAL(EXPT(10, rV-10));
        IG.eState := Valid;
        IG.xPRESS_OK := TRUE; //Backwards compatibility
    ELSIF rV > 8.7 AND rV < 10 THEN
        IG.rPRESS :=rOffPressure;
        IG.xPRESS_OK := FALSE;
        IG.eState := Off;
    ELSE
        IG.rPRESS := rOffPressure;
        IG.xPRESS_OK := FALSE;
        IG.eState := OoR;
    END_IF
ELSE
    IG.rPRESS := rOffPressure;
    IG.xPRESS_OK := FALSE;
    IG.eState := GaugeDisconnected;
END_IF


IF (PG.rPRESS <= IG.rPRO_SP)  AND (PG.xPRESS_OK) THEN
         IG.q_xHV_DIS := IG.xHV_SW;
         IG.xILKOk := TRUE;
    ELSIF NOT IG.q_xHV_DIS AND timer.Q THEN
        IF IG.rPRESS > (IG.rPRO_SP + IG.rHYS_PR) OR PG.rPRESS > (IG.rPRO_SP + IG.rHYS_PR) THEN
        IG.q_xHV_DIS := FALSE;
        IG.xHV_SW := FALSE;
        END_IF
    ELSE
        IG.q_xHV_DIS := FALSE;
        IG.xHV_SW := FALSE;
        IG.xILKOk := FALSE;
     END_IF


timer(IN:= NOT IG.q_xHV_DIS, PT:= T#2s);

(* Setpoint evaluation *)
IG.xAT_VAC := IG.xPRESS_OK AND (IG.rPRESS < IG.rVAC_SP);

(*Soft IO Mapping*)
ACT_IO();
(*Load or save the persistent variables*)
ACT_Persistent();

(*Logger*)
THIS^.ACT_Logger();

(*Load or save the persistent variables*)
ACT_Persistent();

ACTION ACT_IO:
(*soft link inputs*)
IG.i_iPRESS_R:=	i_iPRESS_R;

(*soft link outputs*)
q_xHV_DIS := IG.q_xHV_DIS;
END_ACTION

ACTION ACT_Logger:
// ILK logger
IF NOT IG.xILKOk AND NOT IG.q_xHV_DIS THEN
         fbLogger(sMsg:='Lost external interlock while gauge was on.', eSevr:=TcEventSeverity.Critical);
END_IF


// Log Action
tAction(CLK:=  IG.q_xHV_DIS);
IF tAction.Q THEN fbLogger(sMsg:='Ion gauge commanded to switch on', eSevr:=TcEventSeverity.Info); END_IF



//STATE Logger
IF ePrevState <> IG.eState THEN
      CASE IG.eState OF
        ValidHi:
        ValidLo:
        Valid:
            fbLogger(sMsg:='Gauge pressure valid.', eSevr:=TcEventSeverity.Info);
          GaugeDisconnected:
            fbLogger(sMsg:='Gauge Disconnected.', eSevr:=TcEventSeverity.Critical);
        PressInvalid:
            fbLogger(sMsg:='Gauge pressure invalid.', eSevr:=TcEventSeverity.Warning);
        OoR:
            fbLogger(sMsg:='Gauge pressure out of range.', eSevr:=TcEventSeverity.Warning);
        Starting:
            fbLogger(sMsg:='Gauge starting.', eSevr:=TcEventSeverity.Info);
      END_CASE
      ePrevState := IG.eState;
END_IF
END_ACTION

ACTION ACT_Persistent:
(*On first PLC pass, load the persistent value into the structrue variable*)
IF (SUPER^.bRestorePersistentData) THEN
    SUPER^.bRestorePersistentData	:= FALSE;
    IF ( rVAC_SP <> 0) THEN
        IG.rVAC_SP := rVAC_SP;
    END_IF;
    IF ( rPRO_SP <> 0) THEN
        IG.rPRO_SP := rPRO_SP;
    END_IF;
    IF ( rHYS_PR <> 0) THEN
        IG.rHYS_PR := rHYS_PR;
    END_IF;
END_IF
(*Check if a new value has been written in the structure variable copy it to the persistent variable*)
IF NOT (IG.rVAC_SP = rVAC_SP)  THEN
    rVAC_SP := IG.rVAC_SP;
END_IF;

IF NOT (IG.rPRO_SP = rPRO_SP) THEN
    rPRO_SP:= IG.rPRO_SP;
END_IF;

IF NOT (IG.rHYS_PR = rHYS_PR) THEN
    rHYS_PR:= IG.rHYS_PR;
END_IF;
END_ACTION

METHOD M_AutoOn : BOOL
VAR_INPUT
END_VAR
this^.IG.q_xHV_DIS:= FALSE;
END_METHOD

METHOD M_SetBits : BOOL
VAR_INPUT
    TermBits : UINT; // The terminal's maximum value in bits
END_VAR
This^.iTermBits := TermBits;
END_METHOD

END_FUNCTION_BLOCK

// ---- POUs/Functions/Gauges/FB_CMR362.TcPOU
(* For Pfeiffer CMR 362 *)
FUNCTION_BLOCK FB_CMR362
VAR_INPUT
END_VAR
VAR_OUTPUT
        {attribute 'pytmc' := 'pv:'}
        PG : ST_VG;
END_VAR
VAR
    MinPressure: REAL := 7.5E-3; //Torr
    FullScale : REAL := 75.0 ; //Torr
    V : REAL;
    iTermBits: UINT := 32767 ; // The terminal's maximum value in bits
    (*IO*)
    i_iPRESS_R AT%I* :INT; // input Pressure // Link to analog Input
END_VAR


(* For Pfeiffer CMR 362 *)
(*Soft IO Mapping*)
ACT_IO();

(* Real-value calculation *)
If (iTermBits=0) THEN iTermBits := 32767;END_IF
V := 10*INT_TO_REAL(PG.i_iPRESS_R)/iTermBits;


IF V < 0.4 THEN

    PG.eState := GaugeDisconnected; //Most likely not connected

ELSIF V >= 0.4 AND V <= 1.0 THEN
    PG.rPRESS := MinPressure;
    PG.eState := ValidLo;

ELSIF V > 1 AND V <= 9.8 THEN

    PG.rPRESS := LREAL_TO_REAL((V-1)*0.125*FullScale);
    PG.eState := Valid;

ELSE

PG.eState := OoR; //Larger voltage, probably out of range?

END_IF


(* Pressure OK check *)
PG.xPRESS_OK := (PG.rPRESS >= MinPressure);

(*Soft IO Mapping*)
ACT_IO();

ACTION ACT_IO:
PG.i_iPRESS_R :=i_iPRESS_R;
END_ACTION

METHOD M_SetBits : BOOL
VAR_INPUT
    TermBits : UINT; // The terminal's maximum value in bits
END_VAR
This^.iTermBits := TermBits;
END_METHOD

END_FUNCTION_BLOCK

// ---- POUs/Functions/Gauges/FB_GCM.TcPOU
(* For Baratron Pressure Gauge *)
(*The full-scale pressure times the ratio of the meas.
voltage to full-scale voltage (10V).
The minimum pressure is always going to be 5e-4 * F.S.V.*)
FUNCTION_BLOCK FB_GCM
VAR_IN_OUT

END_VAR
VAR_OUTPUT
    {attribute 'pytmc' := 'pv:'}
    PG	:	ST_VG;
END_VAR
VAR_INPUT
    i_rFULL_SCALE : REAL;
END_VAR
VAR
    rMinPressure: REAL;
    rHYST_PERC	:	REAL := 0.80;	// Hysteresis percentage
    rV	:REAL;
    iTermBits: UINT := 32767 ; // The terminal's maximum value in bits
    (*IO*)
    i_iPRESS_R AT%I* :INT; // input Pressure // Link to analog Input
END_VAR

(* Baratron Pressure Calc
A. Wallace
2016-6-16
The full-scale pressure times the ratio of the meas.
voltage to full-scale voltage (10V).
The minimum pressure is always going to be 5e-4 * F.S.V.*)
PG.rFULL_SCALE := i_rFULL_SCALE;
rMinPressure := PG.rFULL_SCALE * 5E-4;

If (iTermBits=0) THEN iTermBits := 32767;END_IF
rV :=MAX((10*INT_TO_REAL(PG.i_iPRESS_R)/iTermBits),0);

PG.rPRESS := (PG.rFULL_SCALE/10)*rV;
IF PG.rPRESS > (rMinPressure)THEN
    PG.xPRESS_OK := TRUE;
    PG.eState := Valid;
ELSE
    PG.xPRESS_OK := FALSE;
    PG.eState := PressInvalid;
END_IF

(*IO soft linking*)
ACT_IO();

ACTION ACT_IO:
PG.i_iPRESS_R :=i_iPRESS_R;
END_ACTION

METHOD M_SetBits : BOOL
VAR_INPUT
    TermBits : UINT; // The terminal's maximum value in bits
END_VAR
This^.iTermBits := TermBits;
END_METHOD

END_FUNCTION_BLOCK

// ---- POUs/Functions/Gauges/FB_ITR90.TcPOU
(* This function block implements the Oerlikon Leybold IONVAC Hot Cathode ITR 90*)
FUNCTION_BLOCK FB_ITR90
VAR_INPUT
END_VAR
VAR_OUTPUT
    {attribute 'pytmc' := '
    pv:
    '}
    PG : ST_VG;
END_VAR
VAR
    rV : REAL;	// input voltage
    rC: REAL := -0.125; // a constant in the manual (pressure unit dependent)
    rK: REAL := 1.0;// Calibration factor C (gas type dependent)
    iTermBits: UINT := 32767 ; // The terminal's maximum value in bits
    (*IO*)
    i_iPRESS_R AT%I* :INT; // input Pressure // Link to analog Input
END_VAR

(* This function block implements the Oerlikon Leybold IONVAC Hot Cathode ITR 90*)

(* Real-value calculation *)

rV := 10*INT_TO_REAL(PG.i_iPRESS_R)/iTermBits;
PG.rPRESS := (LREAL_TO_REAL(EXPT(10,(rV-7.75)/0.75+rC))) * rK;


(* Pressure gauge State checks *)

//IF (rV <=9.7 ) AND (rV>=1) THEN
    //PG.eState := Valid; // normal
IF rV >= 0.5 AND rV <= 4.5 THEN
    PG.eState := ValidLo; //LO
ELSIF rV > 4.5 AND rV<= 9.9 THEN
    PG.eState := ValidHi; //HIGH
ELSIF rV < 0.5 THEN
    PG.eState := GaugeDisconnected; //not on
ELSE
    PG.eState := PressInvalid; //other fault - could be no gauge, controller powering up etc
END_IF



(* Pressure gauge OK checks *)
PG.xPRESS_OK := (rV <=9.9 ) AND (rV>=0.5);


(* Setpoint evaluation *)
PG.xAT_VAC := PG.xPRESS_OK AND PG.rPRESS < PG.rVAC_SP;


(*Soft IO Linking*)
ACT_IO();

ACTION ACT_IO:
PG.i_iPRESS_R :=i_iPRESS_R;
END_ACTION

METHOD M_SetBits : BOOL
VAR_INPUT
    TermBits : UINT; // The terminal's maximum value in bits
END_VAR
If (iTermBits=0) THEN iTermBits := 32767;END_IF
This^.iTermBits := TermBits;
END_METHOD

END_FUNCTION_BLOCK

// ---- POUs/Functions/Gauges/FB_MKS392.TcPOU
(* This function block implements the MKS392 gauge*)
FUNCTION_BLOCK FB_MKS392
VAR_INPUT
END_VAR
VAR_OUTPUT
    {attribute 'pytmc' := '
    pv:
    '}
    PG : ST_VG;
END_VAR
VAR
    rV : REAL;	// input voltage
    iTermBits: UINT := 32767 ; // The terminal's maximum value in bits
    (*IO*)
    i_iPRESS_R AT%I* :INT; // input Pressure // Link to analog Input
END_VAR

(* Real-value calculation *)
rV := 10*INT_TO_REAL(PG.i_iPRESS_R)/iTermBits;
PG.rPRESS := (LREAL_TO_REAL(EXPT(10,(2*rV)-11)));


(* Pressure gauge State checks *)

IF rV >= 0.5 AND rV <= 3.5 THEN
    PG.eState := ValidLo; //LO
ELSIF rV > 3.5 AND rV<= 6.5 THEN
    PG.eState := ValidHi; //HIGH
ELSIF rV < 0.5 THEN
    PG.eState := GaugeDisconnected; //not on
ELSE
    PG.eState := PressInvalid; //other fault - could be no gauge, controller powering up etc
END_IF



(* Pressure gauge OK checks *)
PG.xPRESS_OK := (rV <=6.5 ) AND (rV>=0.5);


(* Setpoint evaluation *)
PG.xAT_VAC := PG.xPRESS_OK AND PG.rPRESS < PG.rVAC_SP;


(*Soft IO Linking*)
ACT_IO();

ACTION ACT_IO:
PG.i_iPRESS_R :=i_iPRESS_R;
END_ACTION

METHOD M_SetBits : BOOL
VAR_INPUT
    TermBits : UINT; // The terminal's maximum value in bits
END_VAR
This^.iTermBits := TermBits;
END_METHOD

END_FUNCTION_BLOCK

// ---- POUs/Functions/Gauges/FB_MKS500.TcPOU
(* This function is for the Cold Cathode MKS 500.

If connected to Beckhoff EP boxes. Set the EP bit to TRUE, this is necessary for the
MKS500-to-EP box interface because the EP boxes do not natively support the 5v IO
signals on the MKS500 gauge.

A setup process is required for the MKS500 to be usable.
See here: https://confluence.slac.stanford.edu/display/PCDS/MKS+500+-+Cold+Cathode

This function provides ILK and Set Point Protection for the Cold Cathode.
*)

FUNCTION_BLOCK FB_MKS500 EXTENDS FB_GaugeBase
VAR_IN_OUT

END_VAR
VAR_INPUT
    PG	:	ST_VG;
    bEP : BOOL :=FALSE; // Set to True if This Gauge is connected to EP BOX and not EL Terminals
    tRecoverDelay:TIME:=T#600S; (*Delay Time after the first cycle to start the device. Default is 600S*)
END_VAR
VAR_OUTPUT
{attribute 'pytmc' := '
    pv:
    '}
    IG : ST_VG;
END_VAR
VAR
    rV : REAL;
    GaugeTurnOnTmr : TON;
    tStartupTimer:TON;
    iTermBits: UINT := 32767 ; // The terminal's maximum value in bits
    (*IOs to be linked*)
    /// Controls and I/Os
    i_iPRESS_R AT %I* :INT; // input Pressure // Link to analog Input
    q_xHV_DIS AT %Q* : BOOL; // Enable High Voltage when True // 'TcLinkTo' (EP2624) ^Output
    // only for EL and ES terminal
    i_xHV_ON AT %I*	: BOOL; //  True when High Voltage is on  // 'TcLinkTo' (EL1124) ^Input
    i_xDisc_Active AT %I* : BOOL;// Discharge Current Active // 'TcLinkTo' (EL1124) ^Input
    binit:BOOL:=TRUE;
END_VAR

VAR CONSTANT
    // Ranges has to match the configurator software
    pBase : REAL :=1.0E-10;//default curve base pressure is 1E-10. Confusing since can't actually read that low using analog out.
    vBase : REAL := 1;
    vDisconnected : REAL:= 0.5;
    vSlope : REAL := 1.0;
    vGaugeOff: REAL := 9.8;
    vNoDischarge: REAL := 9.3;
    MinPressure: REAL := 1E-10;
    cDefaultPressure : REAL := 0;
    rDeadband : REAL :=0.3;
END_VAR
VAR PERSISTENT
    bWasOn : BOOL;
    bAutoRecover:BOOL;
    bAutoRecoverWrite:BOOL;
END_VAR

(*Startup time*)
IF (bInit) THEN
    tStartupTimer.IN:=TRUE;
    bInit :=FALSE;
END_IF
tStartupTimer(PT:=T#3S);

(* 500 Logarithmic Output Conversion, factory default configuration *)
If (iTermBits=0) THEN iTermBits := 32767;END_IF
rV := 10*INT_TO_REAL(IG.i_iPRESS_R)/iTermBits;

(* Set Guage State based on the Analog voltage*)
IF  NOT (tStartupTimer.Q) THEN // Give time for the gauge controller to start
    IG.eState := Off;
    IG.rPRESS := cDefaultPressure;
ELSIF rV < vDisconnected THEN
    IG.eState := GaugeDisconnected;
    IG.rPRESS := cDefaultPressure;
ELSIF rV >= vDisconnected AND rV < (vNoDischarge -rDeadband)  AND (IG.xHV_SW) THEN
    IG.eState := Valid;
    IG.rPRESS := LREAL_TO_REAL(EXPT(10,((rV-vBase)/vSlope+LOG(pBase))));
ELSIF rV >= (vNoDischarge -rDeadband) AND rV <(vGaugeOff -rDeadband) AND (IG.xHV_SW)  THEN
    IG.eState := Starting;
    IG.rPRESS := LREAL_TO_REAL(EXPT(10,((rV-vBase)/vSlope+LOG(pBase))));
ELSIF rV >= (vGaugeOff -rDeadband) THEN
    IG.eState := Off;
    //IG.rPRESS := LREAL_TO_REAL(EXPT(10,((rV-vBase)/vSlope+LOG(pBase))));
    IG.rPRESS := cDefaultPressure;
ELSIF IG.rPRESS < MinPressure THEN
    IG.eState := PressInvalid;
    //IG.rPRESS := LREAL_TO_REAL(EXPT(10,((rV-vBase)/vSlope+LOG(pBase))));
    IG.rPRESS := cDefaultPressure;
END_IF

(* Set Guage State based on the inputs HV ON and Discharge current*)
If (NOT bEP) THEN
    IF IG.i_xHV_ON AND NOT IG.i_xDisc_Active THEN
        IG.eState := Starting;
        IG.rPRESS := LREAL_TO_REAL(EXPT(10,((rV-vBase)/vSlope+LOG(pBase))));
    ELSIF IG.i_xHV_ON AND IG.i_xDisc_Active THEN
        IG.eState := Valid;
        IG.rPRESS := LREAL_TO_REAL(EXPT(10,((rV-vBase)/vSlope+LOG(pBase))));
    ELSIF NOT IG.i_xHV_ON AND NOT IG.i_xDisc_Active THEN
        IG.eState := Off;
        IG.rPRESS := cDefaultPressure;
    END_IF
END_IF

(* Ion Gauge Protection Functions *)
(* If the PG pressure is greater than the VG.PRO_SP then the gauge is disabled *)
(* If the PG pressure is less than the VG.PRO_SP then the gauge is enabled *)
(* This FB also implements some hysteresis so the gauge doesn't have rapid power cycling while near the turn on boundary *)


IF PG.rPRESS <= IG.rPRO_SP AND PG.xPRESS_OK THEN
    IG.q_xHV_DIS := IG.xHV_SW;
    IG.xILKOk := TRUE;
ELSIF IG.q_xHV_DIS THEN
    IF IG.rPRESS > (IG.rPRO_SP + IG.rHYS_PR)  OR PG.rPRESS > (IG.rPRO_SP + IG.rHYS_PR) THEN
        IG.q_xHV_DIS := FALSE;
        IG.xHV_SW := FALSE;
    END_IF
ELSE
    IG.q_xHV_DIS := FALSE;
    IG.xHV_SW := FALSE;
    IG.xILKOk := FALSE;
END_IF

(* Pressure gauge OK checks *)

GaugeTurnOnTmr(IN:=IG.q_xHV_DIS, PT:=T#10S, Q=>IG.xTurnOnTime);


//Backwards compatibility
IG.xPRESS_OK := (IG.eState = Valid) OR IG.xBAKEOUT;

(* Setpoint evaluation *)
IG.xAT_VAC := (IG.xPRESS_OK AND (IG.rPRESS < IG.rVAC_SP)) OR IG.xBAKEOUT AND (IG.eState = Valid) ;

ACT_Logger();
(*Soft IO Linking*)
// check ethercat Diagnostics
IO();
(*Load or save the persistent variables*)
ACT_Persistent();
(*Run Auto Recovery*)
ACT_Recover();

ACTION ACT_Logger:
// ILK logger
IF (IG.xLog) THEN
    IF NOT IG.xILKOk AND IG.q_xHV_DIS THEN
            fbLogger(sMsg:='Lost external interlock while gauge was on.', eSevr:=TcEventSeverity.Critical);
    END_IF


    // Log Action
    tAction(CLK:=   IG.xHV_SW);
    IF tAction.Q THEN fbLogger(sMsg:='Ion gauge commanded to switch on', eSevr:=TcEventSeverity.Info); END_IF



    //STATE Logger
    tState(CLK:=  ePrevState <> IG.eState);
    IF ePrevState <> IG.eState THEN
          CASE IG.eState OF
            ValidHi:
                fbLogger(sMsg:='Gauge pressure valid high.', eSevr:=TcEventSeverity.Info);
            ValidLo:
                fbLogger(sMsg:='Gauge pressure valid low.', eSevr:=TcEventSeverity.Info);
            Valid:
                fbLogger(sMsg:='Gauge pressure valid.', eSevr:=TcEventSeverity.Info);
            GaugeDisconnected:
                fbLogger(sMsg:='Gauge Disconnected.', eSevr:=TcEventSeverity.Critical);
            PressInvalid:
                fbLogger(sMsg:='Gauge pressure invalid.', eSevr:=TcEventSeverity.Warning);
            OoR:
                fbLogger(sMsg:='Gauge pressure out of range.', eSevr:=TcEventSeverity.Warning);
            Starting:
                fbLogger(sMsg:='Gauge starting.', eSevr:=TcEventSeverity.Info);
          END_CASE
          ePrevState := IG.eState;
          stateTimer.IN := TRUE;
      END_IF
END_IF
END_ACTION

ACTION ACT_Persistent:
(*On first PLC pass, load the persistent value into the structrue variable*)
IF (SUPER^.bRestorePersistentData) THEN
    SUPER^.bRestorePersistentData	:= FALSE;
    IF ( rVAC_SP <> 0) THEN
        IG.rVAC_SP := rVAC_SP;
    END_IF;
    IF ( rPRO_SP <> 0) THEN
        IG.rPRO_SP := rPRO_SP;
    END_IF;
    IF ( rHYS_PR <> 0) THEN
        IG.rHYS_PR := rHYS_PR;
    END_IF;
    IF ( bAutoRecoverWrite) THEN
        IG.xAutoOn := bAutoRecover;
    END_IF;
END_IF
(*Check if a new value has been written in the structure variable copy it to the persistent variable*)
IF NOT (IG.rVAC_SP = rVAC_SP)  THEN
    rVAC_SP := IG.rVAC_SP;
END_IF;

IF NOT (IG.rPRO_SP = rPRO_SP) THEN
    rPRO_SP:= IG.rPRO_SP;
END_IF;

IF NOT (IG.rHYS_PR = rHYS_PR) THEN
    rHYS_PR:= IG.rHYS_PR;
END_IF;

IF NOT(bAutoRecoverWrite) OR NOT (bAutoRecover = IG.xAutoOn) THEN
    bAutoRecover := IG.xAutoOn;
    bAutoRecoverWrite := TRUE;
END_IF;
stateTimer(PT:=T#10S);
IF (stateTimer.Q) THEN
    bWasOn := (IG.eState >=Valid );
    stateTimer.IN := FALSE;
    fbWritePersistentData(NETID:='', PORT:=851, START:=TRUE, TMOUT:=T#1s );
END_IF;
END_ACTION

ACTION ACT_Recover:
fbGetCurTaskIdx();
IF (TwinCAT_SystemInfoVarList._TaskInfo[fbGetCurTaskIdx.index].FirstCycle) THEN
    tRecover.IN := TRUE;
END_IF
tRecover(IN:= , PT:=tRecoverDelay);
IF NOT(bAutoRecoverWrite) OR (tRecover.Q AND bAutoRecover ) THEN
    This^.M_Recover();
    tRecover.IN := FALSE;
END_IF
END_ACTION

ACTION IO:
(*soft link inputs*)
IG.i_iPRESS_R:=	i_iPRESS_R;
IG.i_xHV_ON:= i_xHV_ON;
IG.i_xDisc_Active:=i_xDisc_Active;
(*soft link outputs*)
q_xHV_DIS := IG.q_xHV_DIS;

IG.sPath := sPath;
IG.iAutoOnTimer:= TIME_TO_INT(tRecover.PT);
END_ACTION

METHOD M_HVE : BOOL
VAR_INPUT
        enable:bool; // set to true to enable, false to disable;
END_VAR

this^.IG.xHV_SW:= enable;
END_METHOD

METHOD M_Recover : BOOL
VAR_INPUT
END_VAR
This^.M_HVE(This^.bWasOn);
M_Recover := bWasOn;
IF (bWasOn) THEN fbLogger(sMsg:='Auto Recovery Initiated.', eSevr:=TcEventSeverity.Info); END_IF;
END_METHOD

METHOD M_SetBits : BOOL
VAR_INPUT
    TermBits : UINT; // The terminal's maximum value in bits
END_VAR
This^.iTermBits := TermBits;
END_METHOD

END_FUNCTION_BLOCK

// ---- POUs/Functions/Gauges/FB_MKS722.TcPOU
(* This function is for the MKS 722*)

FUNCTION_BLOCK FB_MKS722
VAR_IN_OUT

END_VAR
VAR_OUTPUT
    {attribute 'pytmc' := '
    pv:
    '}
    VG	:	ST_VG;
END_VAR
VAR_INPUT
    i_rMinPressure	:	REAL;
    i_rMaxPressure	:	REAL;
END_VAR
VAR
    iTermBits: UINT := 32767 ; // The terminal's maximum value in bits
    rMinPressure: REAL;
    rVMin	:	REAL := 0.01; // Anything less than this voltage is considered disconnected
    rVMax :	REAL := 10.5; // Anything more than this is considered invalid
    rV	:REAL;

    (*IO*)
    i_iPRESS_R AT%I* :INT; // input Pressure // Link to analog Input
END_VAR



(* Real-value calculation *)
If (iTermBits=0) THEN iTermBits := 32767;END_IF
rV := 10*INT_TO_REAL(VG.i_iPRESS_R)/iTermBits;


// Is the gauge plugged in, and within a reasonable range?
IF rV < rVMin THEN
    VG.eState := GaugeDisconnected;
ELSIF rV > rVMax THEN
    VG.eState := PressInvalid;
ELSIF VG.rPRESS >= rMinPressure AND VG.rPRESS <= i_rMaxPressure THEN
                VG.eState := Valid;
ELSIF VG.rPRESS < i_rMinPressure THEN
                VG.eState := ValidLo;
ELSE
                VG.eState := ValidHi;
END_IF

// Legacy Press OK boolean eval
VG.xPRESS_OK := VG.eState >= gc_GaugeValidState;

(*IO Soft Mapping*)
ACT_IO();

ACTION ACT_IO:
VG.i_iPRESS_R :=i_iPRESS_R;
END_ACTION

END_FUNCTION_BLOCK

// ---- POUs/Functions/Gauges/FB_MKS_937A.TcPOU
(* 937A Logarithmic Output Conversion *)
(* 7-15-2015 *)
(* This function will read the pressure from any gauge on a 937A. *)
(* To be used when the specific device function block is not available *)
FUNCTION_BLOCK FB_MKS_937A
VAR_IN_OUT

END_VAR
VAR_INPUT
    PG	:	ST_VG := g_DummyVG; // Gauge Structure used to Interlock the ion gauges
END_VAR
VAR_OUTPUT
    {attribute 'pytmc' := 'pv: '}
    VG : ST_VG; // Vacuum Gauge Data Structure
END_VAR
VAR
    rV	:	REAL;
        (*IOs to be linked*)
    /// Controls and I/Os
    i_iPRESS_R AT %I* :INT; // input Pressure // Link to analog Input
    q_xHV_DIS AT %Q* : BOOL; // Disable Gauge High Voltage when True // 'TcLinkTo' (EL2794) ^Output

END_VAR

(* 937A Logarithmic Output Conversion *)
(* 7-15-2015 *)
(* This function will read the pressure from any gauge on a 937A. *)

rV := 10*INT_TO_REAL(VG.i_iPRESS_R)/32767;
VG.rPRESS := LREAL_TO_REAL(EXPT(10,rV/0.6-12));


(* Ion Gauge Protection Functions *)
(* If the PG pressure is greater than the VG.PRO_SP then the gauge is disabled *)
(* If the PG pressure is less than the VG.PRO_SP then the gauge is enabled *)
(* This FB also implements some hysteresis so the gauge doesn't have rapid power cycling while near the turn on boundary *)

IF PG.rPRESS < VG.rPRO_SP THEN

VG.q_xHV_DIS :=  NOT VG.xHV_SW;

ELSIF NOT VG.q_xHV_DIS THEN
    IF VG.rPRESS > VG.rPRO_SP + VG.rHYS_PR OR PG.rPRESS > VG.rPRO_SP + VG.rHYS_PR THEN
        VG.q_xHV_DIS := TRUE;
    END_IF
ELSE
    VG.q_xHV_DIS := TRUE;
END_IF


(* Pressure gauge OK checks *)
VG.xPRESS_OK := (rV <=9.6 ) AND (rV>=0.6); //legacy

IF (rV <=9.6 ) AND (rV>=0.6) THEN
    VG.eState := Valid; // normal
ELSIF rV >= 0.18 AND rV <= 0.22 THEN
    VG.eState := ValidLo; //LO
ELSIF rV >= 9.7 AND rV<= 9.9 THEN
    VG.eState := ValidHi; //HIGH
ELSIF rV < 0.18 THEN
    VG.eState := GaugeDisconnected; //not on
ELSE
    VG.eState := PressInvalid; //other fault - could be no gauge, controller powering up etc
END_IF

(* Setpoint evaluation *)
VG.xAT_VAC := (VG.eState =Valid) AND VG.rPRESS < VG.rVAC_SP;

(*Soft IO Linking*)
ACT_IO();

ACTION ACT_IO:
(*soft link inputs*)
VG.i_iPRESS_R:=	i_iPRESS_R;

(*soft link outputs*)
q_xHV_DIS := VG.q_xHV_DIS;
END_ACTION

END_FUNCTION_BLOCK

